LIN {X 30.043,Y -44.102,Z -90.850,A -90.000,B 90.000,C 0.000} C_DIS
LIN {X 31.596,Y -44.132,Z -91.106,A -90.000,B 90.000,C 0.000} C_DIS
LIN {X 31.805,Y -44.138,Z -91.148,A -90.000,B 90.000,C 0.000} C_DIS
LIN {X 31.963,Y -44.144,Z -91.180,A -90.000,B 90.000,C 0.000} C_DIS
LIN {X 32.126,Y -44.146,Z -91.221,A -90.000,B 90.000,C 0.000} C_DIS
LIN {X 33.590,Y -44.179,Z -91.628,A -90.000,B 90.000,C 0.000} C_DIS
LIN {X 33.752,Y -44.184,Z -91.677,A -90.000,B 90.000,C 0.000} C_DIS
LIN {X 33.947,Y -44.192,Z -91.742,A -90.000,B 90.000,C 0.000} C_DIS
LIN {X 34.606,Y -44.214,Z -91.970,A -90.000,B 90.000,C 0.000} C_DIS
LIN {X 35.661,Y -44.230,Z -92.339,A -90.000,B 90.000,C 0.000} C_DIS
LIN {X 35.939,Y -44.232,Z -92.438,A -90.000,B 90.000,C 0.000} C_DIS
LIN {X 36.161,Y -44.234,Z -92.528,A -90.000,B 90.000,C 0.000} C_DIS
LIN {X 36.724,Y -44.246,Z -92.772,A -90.000,B 90.000,C 0.000} C_DIS
LIN {X 36.900,Y -44.250,Z -92.851,A -90.000,B 90.000,C 0.000} C_DIS
LIN {X 37.063,Y -44.253,Z -92.930,A -90.000,B 90.000,C 0.000} C_DIS
LIN {X 37.996,Y -44.267,Z -93.435,A -90.000,B 90.000,C 0.000} C_DIS
LIN {X 38.705,Y -44.281,Z -93.837,A -90.000,B 90.000,C 0.000} C_DIS
LIN {X 39.137,Y -44.293,Z -94.082,A -90.000,B 90.000,C 0.000} C_DIS
LIN {X 39.281,Y -44.294,Z -94.165,A -90.000,B 90.000,C 0.000} C_DIS
LIN {X 39.455,Y -44.293,Z -94.272,A -90.000,B 90.000,C 0.000} C_DIS
LIN {X 40.133,Y -44.291,Z -94.711,A -90.000,B 90.000,C 0.000} C_DIS
LIN {X 40.366,Y -44.293,Z -94.872,A -90.000,B 90.000,C 0.000} C_DIS
LIN {X 40.619,Y -44.297,Z -95.057,A -90.000,B 90.000,C 0.000} C_DIS
LIN {X 40.830,Y -44.305,Z -95.230,A -90.000,B 90.000,C 0.000} C_DIS
LIN {X 41.144,Y -44.315,Z -95.490,A -90.000,B 90.000,C 0.000} C_DIS
LIN {X 41.855,Y -44.317,Z -96.085,A -90.000,B 90.000,C 0.000} C_DIS
LIN {X 42.021,Y -44.319,Z -96.232,A -90.000,B 90.000,C 0.000} C_DIS
LIN {X 42.450,Y -44.332,Z -96.645,A -90.000,B 90.000,C 0.000} C_DIS
LIN {X 42.787,Y -44.333,Z -96.974,A -90.000,B 90.000,C 0.000} C_DIS
LIN {X 42.967,Y -44.330,Z -97.150,A -90.000,B 90.000,C 0.000} C_DIS
LIN {X 43.705,Y -44.300,Z -97.883,A -90.000,B 90.000,C 0.000} C_DIS
LIN {X 43.789,Y -44.297,Z -97.971,A -90.000,B 90.000,C 0.000} C_DIS
LIN {X 44.031,Y -44.292,Z -98.239,A -90.000,B 90.000,C 0.000} C_DIS
LIN {X 44.098,Y -44.291,Z -98.318,A -90.000,B 90.000,C 0.000} C_DIS
LIN {X 44.222,Y -44.291,Z -98.469,A -90.000,B 90.000,C 0.000} C_DIS
LIN {X 44.387,Y -44.294,Z -98.687,A -90.000,B 90.000,C 0.000} C_DIS
LIN {X 44.481,Y -44.298,Z -98.827,A -90.000,B 90.000,C 0.000} C_DIS
LIN {X 44.610,Y -44.300,Z -99.041,A -90.000,B 90.000,C 0.000} C_DIS
LIN {X 44.729,Y -44.303,Z -99.246,A -90.000,B 90.000,C 0.000} C_DIS
LIN {X 45.134,Y -44.318,Z -99.976,A -90.000,B 90.000,C 0.000} C_DIS
LIN {X 45.262,Y -44.320,Z -100.209,A -90.000,B 90.000,C 0.000} C_DIS
LIN {X 45.761,Y -44.295,Z -101.133,A -90.000,B 90.000,C 0.000} C_DIS
LIN {X 45.808,Y -44.294,Z -101.226,A -90.000,B 90.000,C 0.000} C_DIS
LIN {X 46.111,Y -44.285,Z -101.863,A -90.000,B 90.000,C 0.000} C_DIS
LIN {X 46.252,Y -44.275,Z -102.164,A -90.000,B 90.000,C 0.000} C_DIS
LIN {X 46.732,Y -44.221,Z -103.202,A -90.000,B 90.000,C 0.000} C_DIS
LIN {X 46.781,Y -44.216,Z -103.318,A -90.000,B 90.000,C 0.000} C_DIS
LIN {X 46.871,Y -44.208,Z -103.549,A -90.000,B 90.000,C 0.000} C_DIS
LIN {X 46.913,Y -44.205,Z -103.666,A -90.000,B 90.000,C 0.000} C_DIS
LIN {X 46.986,Y -44.201,Z -103.892,A -90.000,B 90.000,C 0.000} C_DIS
LIN {X 47.046,Y -44.199,Z -104.098,A -90.000,B 90.000,C 0.000} C_DIS
LIN {X 47.095,Y -44.201,Z -104.309,A -90.000,B 90.000,C 0.000} C_DIS
LIN {X 47.115,Y -44.202,Z -104.397,A -90.000,B 90.000,C 0.000} C_DIS
LIN {X 47.180,Y -44.202,Z -104.648,A -90.000,B 90.000,C 0.000} C_DIS
LIN {X 47.223,Y -44.202,Z -104.839,A -90.000,B 90.000,C 0.000} C_DIS
LIN {X 47.252,Y -44.203,Z -104.996,A -90.000,B 90.000,C 0.000} C_DIS
LIN {X 47.278,Y -44.207,Z -105.181,A -90.000,B 90.000,C 0.000} C_DIS
LIN {X 47.321,Y -44.218,Z -105.570,A -90.000,B 90.000,C 0.000} C_DIS
LIN {X 47.363,Y -44.223,Z -106.056,A -90.000,B 90.000,C 0.000} C_DIS
LIN {X 47.384,Y -44.224,Z -106.317,A -90.000,B 90.000,C 0.000} C_DIS
LIN {X 47.440,Y -44.195,Z -107.093,A -90.000,B 90.000,C 0.000} C_DIS
LIN {X 47.552,Y -44.143,Z -108.663,A -90.000,B 90.000,C 0.000} C_DIS
LIN {X 47.559,Y -44.140,Z -108.785,A -90.000,B 90.000,C 0.000} C_DIS
LIN {X 47.562,Y -44.138,Z -108.944,A -90.000,B 90.000,C 0.000} C_DIS
LIN {X 47.556,Y -44.137,Z -109.182,A -90.000,B 90.000,C 0.000} C_DIS
LIN {X 47.550,Y -44.139,Z -109.300,A -90.000,B 90.000,C 0.000} C_DIS
LIN {X 47.472,Y -44.157,Z -110.305,A -90.000,B 90.000,C 0.000} C_DIS
LIN {X 47.309,Y -44.112,Z -112.094,A -90.000,B 90.000,C 0.000} C_DIS
LIN {X 47.205,Y -44.092,Z -113.075,A -90.000,B 90.000,C 0.000} C_DIS
LIN {X 47.187,Y -44.091,Z -113.203,A -90.000,B 90.000,C 0.000} C_DIS
LIN {X 47.137,Y -44.091,Z -113.498,A -90.000,B 90.000,C 0.000} C_DIS
LIN {X 47.119,Y -44.093,Z -113.585,A -90.000,B 90.000,C 0.000} C_DIS
LIN {X 47.045,Y -44.099,Z -113.899,A -90.000,B 90.000,C 0.000} C_DIS
LIN {X 46.943,Y -44.102,Z -114.328,A -90.000,B 90.000,C 0.000} C_DIS
LIN {X 46.601,Y -44.049,Z -115.684,A -90.000,B 90.000,C 0.000} C_DIS
LIN {X 46.560,Y -44.044,Z -115.831,A -90.000,B 90.000,C 0.000} C_DIS
LIN {X 46.147,Y -44.010,Z -117.234,A -90.000,B 90.000,C 0.000} C_DIS
LIN {X 46.088,Y -44.008,Z -117.419,A -90.000,B 90.000,C 0.000} C_DIS
LIN {X 45.995,Y -44.008,Z -117.676,A -90.000,B 90.000,C 0.000} C_DIS
LIN {X 45.962,Y -44.009,Z -117.763,A -90.000,B 90.000,C 0.000} C_DIS
LIN {X 45.889,Y -44.013,Z -117.937,A -90.000,B 90.000,C 0.000} C_DIS
LIN {X 45.762,Y -44.020,Z -118.219,A -90.000,B 90.000,C 0.000} C_DIS
LIN {X 45.357,Y -43.999,Z -119.084,A -90.000,B 90.000,C 0.000} C_DIS
LIN {X 45.158,Y -43.991,Z -119.498,A -90.000,B 90.000,C 0.000} C_DIS
LIN {X 44.451,Y -43.966,Z -120.974,A -90.000,B 90.000,C 0.000} C_DIS
LIN {X 44.317,Y -43.963,Z -121.251,A -90.000,B 90.000,C 0.000} C_DIS
LIN {X 44.210,Y -43.963,Z -121.454,A -90.000,B 90.000,C 0.000} C_DIS
LIN {X 44.078,Y -43.968,Z -121.683,A -90.000,B 90.000,C 0.000} C_DIS
LIN {X 43.957,Y -43.966,Z -121.881,A -90.000,B 90.000,C 0.000} C_DIS
LIN {X 43.022,Y -43.933,Z -123.308,A -90.000,B 90.000,C 0.000} C_DIS
LIN {X 42.446,Y -43.896,Z -124.174,A -90.000,B 90.000,C 0.000} C_DIS
LIN {X 42.367,Y -43.892,Z -124.288,A -90.000,B 90.000,C 0.000} C_DIS
LIN {X 41.848,Y -43.874,Z -125.016,A -90.000,B 90.000,C 0.000} C_DIS
LIN {X 41.755,Y -43.871,Z -125.141,A -90.000,B 90.000,C 0.000} C_DIS
LIN {X 40.950,Y -43.838,Z -126.136,A -90.000,B 90.000,C 0.000} C_DIS
LIN {X 40.132,Y -43.777,Z -127.128,A -90.000,B 90.000,C 0.000} C_DIS
LIN {X 39.865,Y -43.763,Z -127.435,A -90.000,B 90.000,C 0.000} C_DIS
LIN {X 39.099,Y -43.739,Z -128.268,A -90.000,B 90.000,C 0.000} C_DIS
LIN {X 38.728,Y -43.722,Z -128.669,A -90.000,B 90.000,C 0.000} C_DIS
LIN {X 38.085,Y -43.674,Z -129.350,A -90.000,B 90.000,C 0.000} C_DIS
LIN {X 37.439,Y -43.621,Z -130.031,A -90.000,B 90.000,C 0.000} C_DIS
LIN {X 37.295,Y -43.613,Z -130.175,A -90.000,B 90.000,C 0.000} C_DIS
LIN {X 36.203,Y -43.578,Z -131.197,A -90.000,B 90.000,C 0.000} C_DIS
LIN {X 35.591,Y -43.550,Z -131.813,A -90.000,B 90.000,C 0.000} C_DIS
LIN {X 34.765,Y -43.481,Z -132.619,A -90.000,B 90.000,C 0.000} C_DIS
LIN {X 34.182,Y -43.434,Z -133.184,A -90.000,B 90.000,C 0.000} C_DIS
LIN {X 34.040,Y -43.425,Z -133.315,A -90.000,B 90.000,C 0.000} C_DIS
LIN {X 32.759,Y -43.384,Z -134.425,A -90.000,B 90.000,C 0.000} C_DIS
LIN {X 31.780,Y -43.308,Z -135.363,A -90.000,B 90.000,C 0.000} C_DIS
LIN {X 31.780,Y -60.000,Z -135.363,A -90.000,B 90.000,C 0.000} C_DIS
LIN {X 27.880,Y -60.000,Z -88.546,A -90.000,B 90.000,C 0.000} C_DIS
LIN {X 27.880,Y -43.308,Z -88.546,A -90.000,B 90.000,C 0.000} C_DIS
LIN {X 28.059,Y -43.318,Z -88.565,A -90.000,B 90.000,C 0.000} C_DIS
LIN {X 28.163,Y -43.325,Z -88.579,A -90.000,B 90.000,C 0.000} C_DIS
LIN {X 28.312,Y -43.338,Z -88.598,A -90.000,B 90.000,C 0.000} C_DIS
LIN {X 28.537,Y -43.361,Z -88.634,A -90.000,B 90.000,C 0.000} C_DIS
LIN {X 29.638,Y -43.432,Z -88.839,A -90.000,B 90.000,C 0.000} C_DIS
LIN {X 30.344,Y -43.470,Z -88.974,A -90.000,B 90.000,C 0.000} C_DIS
LIN {X 30.370,Y -43.472,Z -88.979,A -90.000,B 90.000,C 0.000} C_DIS
LIN {X 31.919,Y -43.541,Z -89.223,A -90.000,B 90.000,C 0.000} C_DIS
LIN {X 32.192,Y -43.555,Z -89.274,A -90.000,B 90.000,C 0.000} C_DIS
LIN {X 32.370,Y -43.563,Z -89.310,A -90.000,B 90.000,C 0.000} C_DIS
LIN {X 32.600,Y -43.574,Z -89.365,A -90.000,B 90.000,C 0.000} C_DIS
LIN {X 34.122,Y -43.639,Z -89.777,A -90.000,B 90.000,C 0.000} C_DIS
LIN {X 34.326,Y -43.649,Z -89.837,A -90.000,B 90.000,C 0.000} C_DIS
LIN {X 34.574,Y -43.663,Z -89.918,A -90.000,B 90.000,C 0.000} C_DIS
LIN {X 34.743,Y -43.669,Z -89.976,A -90.000,B 90.000,C 0.000} C_DIS
LIN {X 36.312,Y -43.705,Z -90.522,A -90.000,B 90.000,C 0.000} C_DIS
LIN {X 36.590,Y -43.708,Z -90.621,A -90.000,B 90.000,C 0.000} C_DIS
LIN {X 36.883,Y -43.714,Z -90.736,A -90.000,B 90.000,C 0.000} C_DIS
LIN {X 37.249,Y -43.714,Z -90.897,A -90.000,B 90.000,C 0.000} C_DIS
LIN {X 37.752,Y -43.711,Z -91.123,A -90.000,B 90.000,C 0.000} C_DIS
LIN {X 37.986,Y -43.719,Z -91.238,A -90.000,B 90.000,C 0.000} C_DIS
LIN {X 38.913,Y -43.761,Z -91.731,A -90.000,B 90.000,C 0.000} C_DIS
LIN {X 38.987,Y -43.763,Z -91.772,A -90.000,B 90.000,C 0.000} C_DIS
LIN {X 39.920,Y -43.783,Z -92.302,A -90.000,B 90.000,C 0.000} C_DIS
LIN {X 40.246,Y -43.784,Z -92.489,A -90.000,B 90.000,C 0.000} C_DIS
LIN {X 40.465,Y -43.786,Z -92.621,A -90.000,B 90.000,C 0.000} C_DIS
LIN {X 40.951,Y -43.795,Z -92.932,A -90.000,B 90.000,C 0.000} C_DIS
LIN {X 41.185,Y -43.792,Z -93.085,A -90.000,B 90.000,C 0.000} C_DIS
LIN {X 41.470,Y -43.790,Z -93.283,A -90.000,B 90.000,C 0.000} C_DIS
LIN {X 41.766,Y -43.790,Z -93.499,A -90.000,B 90.000,C 0.000} C_DIS
LIN {X 41.857,Y -43.790,Z -93.570,A -90.000,B 90.000,C 0.000} C_DIS
LIN {X 42.397,Y -43.801,Z -94.019,A -90.000,B 90.000,C 0.000} C_DIS
LIN {X 42.561,Y -43.807,Z -94.153,A -90.000,B 90.000,C 0.000} C_DIS
LIN {X 42.874,Y -43.816,Z -94.412,A -90.000,B 90.000,C 0.000} C_DIS
LIN {X 43.145,Y -43.817,Z -94.640,A -90.000,B 90.000,C 0.000} C_DIS
LIN {X 43.339,Y -43.815,Z -94.815,A -90.000,B 90.000,C 0.000} C_DIS
LIN {X 44.418,Y -43.818,Z -95.866,A -90.000,B 90.000,C 0.000} C_DIS
LIN {X 44.651,Y -43.815,Z -96.094,A -90.000,B 90.000,C 0.000} C_DIS
LIN {X 45.058,Y -43.797,Z -96.498,A -90.000,B 90.000,C 0.000} C_DIS
LIN {X 45.182,Y -43.793,Z -96.627,A -90.000,B 90.000,C 0.000} C_DIS
LIN {X 45.463,Y -43.786,Z -96.938,A -90.000,B 90.000,C 0.000} C_DIS
LIN {X 45.596,Y -43.784,Z -97.094,A -90.000,B 90.000,C 0.000} C_DIS
LIN {X 45.754,Y -43.783,Z -97.288,A -90.000,B 90.000,C 0.000} C_DIS
LIN {X 45.968,Y -43.786,Z -97.573,A -90.000,B 90.000,C 0.000} C_DIS
LIN {X 46.087,Y -43.783,Z -97.752,A -90.000,B 90.000,C 0.000} C_DIS
LIN {X 46.267,Y -43.781,Z -98.049,A -90.000,B 90.000,C 0.000} C_DIS
LIN {X 46.405,Y -43.780,Z -98.288,A -90.000,B 90.000,C 0.000} C_DIS
LIN {X 47.442,Y -43.730,Z -100.210,A -90.000,B 90.000,C 0.000} C_DIS
LIN {X 47.514,Y -43.727,Z -100.349,A -90.000,B 90.000,C 0.000} C_DIS
LIN {X 48.139,Y -43.712,Z -101.661,A -90.000,B 90.000,C 0.000} C_DIS
LIN {X 48.380,Y -43.693,Z -102.177,A -90.000,B 90.000,C 0.000} C_DIS
LIN {X 48.470,Y -43.682,Z -102.371,A -90.000,B 90.000,C 0.000} C_DIS
LIN {X 48.568,Y -43.669,Z -102.606,A -90.000,B 90.000,C 0.000} C_DIS
LIN {X 48.643,Y -43.653,Z -102.804,A -90.000,B 90.000,C 0.000} C_DIS
LIN {X 48.715,Y -43.636,Z -103.011,A -90.000,B 90.000,C 0.000} C_DIS
LIN {X 48.803,Y -43.616,Z -103.296,A -90.000,B 90.000,C 0.000} C_DIS
LIN {X 48.876,Y -43.601,Z -103.555,A -90.000,B 90.000,C 0.000} C_DIS
LIN {X 48.905,Y -43.595,Z -103.673,A -90.000,B 90.000,C 0.000} C_DIS
LIN {X 48.958,Y -43.586,Z -103.919,A -90.000,B 90.000,C 0.000} C_DIS
LIN {X 49.017,Y -43.574,Z -104.168,A -90.000,B 90.000,C 0.000} C_DIS
LIN {X 49.083,Y -43.562,Z -104.475,A -90.000,B 90.000,C 0.000} C_DIS
LIN {X 49.116,Y -43.558,Z -104.663,A -90.000,B 90.000,C 0.000} C_DIS
LIN {X 49.152,Y -43.556,Z -104.928,A -90.000,B 90.000,C 0.000} C_DIS
LIN {X 49.200,Y -43.558,Z -105.382,A -90.000,B 90.000,C 0.000} C_DIS
LIN {X 49.314,Y -43.572,Z -106.702,A -90.000,B 90.000,C 0.000} C_DIS
LIN {X 49.338,Y -43.572,Z -106.983,A -90.000,B 90.000,C 0.000} C_DIS
LIN {X 49.445,Y -43.516,Z -108.506,A -90.000,B 90.000,C 0.000} C_DIS
LIN {X 49.454,Y -43.501,Z -108.743,A -90.000,B 90.000,C 0.000} C_DIS
LIN {X 49.455,Y -43.493,Z -108.912,A -90.000,B 90.000,C 0.000} C_DIS
LIN {X 49.446,Y -43.483,Z -109.215,A -90.000,B 90.000,C 0.000} C_DIS
LIN {X 49.435,Y -43.479,Z -109.402,A -90.000,B 90.000,C 0.000} C_DIS
LIN {X 49.294,Y -43.461,Z -111.026,A -90.000,B 90.000,C 0.000} C_DIS
LIN {X 49.267,Y -43.452,Z -111.313,A -90.000,B 90.000,C 0.000} C_DIS
LIN {X 49.173,Y -43.402,Z -112.245,A -90.000,B 90.000,C 0.000} C_DIS
LIN {X 49.055,Y -43.354,Z -113.257,A -90.000,B 90.000,C 0.000} C_DIS
LIN {X 49.016,Y -43.344,Z -113.516,A -90.000,B 90.000,C 0.000} C_DIS
LIN {X 48.949,Y -43.336,Z -113.881,A -90.000,B 90.000,C 0.000} C_DIS
LIN {X 48.918,Y -43.336,Z -114.020,A -90.000,B 90.000,C 0.000} C_DIS
LIN {X 48.648,Y -43.340,Z -115.154,A -90.000,B 90.000,C 0.000} C_DIS
LIN {X 48.456,Y -43.308,Z -115.911,A -90.000,B 90.000,C 0.000} C_DIS
LIN {X 48.456,Y -60.000,Z -115.911,A -90.000,B 90.000,C 0.000} C_DIS
LIN {X 43.124,Y -60.000,Z -92.100,A -90.000,B 90.000,C 0.000} C_DIS
LIN {X 43.124,Y -43.308,Z -92.100,A -90.000,B 90.000,C 0.000} C_DIS
LIN {X 43.760,Y -43.320,Z -92.627,A -90.000,B 90.000,C 0.000} C_DIS
LIN {X 44.439,Y -43.322,Z -93.197,A -90.000,B 90.000,C 0.000} C_DIS
LIN {X 44.570,Y -43.324,Z -93.315,A -90.000,B 90.000,C 0.000} C_DIS
LIN {X 44.698,Y -43.320,Z -93.434,A -90.000,B 90.000,C 0.000} C_DIS
LIN {X 45.276,Y -43.308,Z -94.001,A -90.000,B 90.000,C 0.000} C_DIS
LIN {X 45.276,Y -60.000,Z -94.001,A -90.000,B 90.000,C 0.000} C_DIS
LIN {X -15.244,Y -60.000,Z -137.680,A -90.000,B 90.000,C 0.000} C_DIS
LIN {X -15.244,Y -43.308,Z -137.680,A -90.000,B 90.000,C 0.000} C_DIS
LIN {X -15.380,Y -43.347,Z -137.361,A -90.000,B 90.000,C 0.000} C_DIS
LIN {X -15.513,Y -43.390,Z -137.028,A -90.000,B 90.000,C 0.000} C_DIS
LIN {X -15.611,Y -43.411,Z -136.767,A -90.000,B 90.000,C 0.000} C_DIS
LIN {X -15.839,Y -43.449,Z -136.149,A -90.000,B 90.000,C 0.000} C_DIS
LIN {X -15.880,Y -43.453,Z -136.030,A -90.000,B 90.000,C 0.000} C_DIS
LIN {X -16.000,Y -43.464,Z -135.661,A -90.000,B 90.000,C 0.000} C_DIS
LIN {X -16.068,Y -43.474,Z -135.427,A -90.000,B 90.000,C 0.000} C_DIS
LIN {X -16.120,Y -43.485,Z -135.220,A -90.000,B 90.000,C 0.000} C_DIS
LIN {X -16.156,Y -43.495,Z -135.060,A -90.000,B 90.000,C 0.000} C_DIS
LIN {X -16.243,Y -43.528,Z -134.606,A -90.000,B 90.000,C 0.000} C_DIS
LIN {X -16.291,Y -43.540,Z -134.342,A -90.000,B 90.000,C 0.000} C_DIS
LIN {X -16.453,Y -43.560,Z -133.399,A -90.000,B 90.000,C 0.000} C_DIS
LIN {X -16.487,Y -43.566,Z -133.170,A -90.000,B 90.000,C 0.000} C_DIS
LIN {X -16.536,Y -43.579,Z -132.789,A -90.000,B 90.000,C 0.000} C_DIS
LIN {X -16.555,Y -43.590,Z -132.587,A -90.000,B 90.000,C 0.000} C_DIS
LIN {X -16.567,Y -43.598,Z -132.329,A -90.000,B 90.000,C 0.000} C_DIS
LIN {X -16.575,Y -43.608,Z -132.021,A -90.000,B 90.000,C 0.000} C_DIS
LIN {X -16.575,Y -43.613,Z -131.842,A -90.000,B 90.000,C 0.000} C_DIS
LIN {X -16.565,Y -43.622,Z -131.524,A -90.000,B 90.000,C 0.000} C_DIS
LIN {X -16.533,Y -43.637,Z -131.071,A -90.000,B 90.000,C 0.000} C_DIS
LIN {X -16.510,Y -43.647,Z -130.766,A -90.000,B 90.000,C 0.000} C_DIS
LIN {X -16.464,Y -43.666,Z -130.269,A -90.000,B 90.000,C 0.000} C_DIS
LIN {X -16.339,Y -43.680,Z -129.038,A -90.000,B 90.000,C 0.000} C_DIS
LIN {X -16.304,Y -43.685,Z -128.769,A -90.000,B 90.000,C 0.000} C_DIS
LIN {X -16.269,Y -43.692,Z -128.557,A -90.000,B 90.000,C 0.000} C_DIS
LIN {X -16.232,Y -43.701,Z -128.334,A -90.000,B 90.000,C 0.000} C_DIS
LIN {X -16.080,Y -43.723,Z -127.467,A -90.000,B 90.000,C 0.000} C_DIS
LIN {X -16.014,Y -43.733,Z -127.175,A -90.000,B 90.000,C 0.000} C_DIS
LIN {X -15.964,Y -43.742,Z -126.978,A -90.000,B 90.000,C 0.000} C_DIS
LIN {X -15.876,Y -43.758,Z -126.673,A -90.000,B 90.000,C 0.000} C_DIS
LIN {X -15.607,Y -43.810,Z -125.802,A -90.000,B 90.000,C 0.000} C_DIS
LIN {X -15.423,Y -43.845,Z -125.098,A -90.000,B 90.000,C 0.000} C_DIS
LIN {X -15.140,Y -43.879,Z -124.031,A -90.000,B 90.000,C 0.000} C_DIS
LIN {X -15.107,Y -43.886,Z -123.903,A -90.000,B 90.000,C 0.000} C_DIS
LIN {X -15.003,Y -43.907,Z -123.535,A -90.000,B 90.000,C 0.000} C_DIS
LIN {X -14.926,Y -43.923,Z -123.288,A -90.000,B 90.000,C 0.000} C_DIS
LIN {X -14.894,Y -43.930,Z -123.197,A -90.000,B 90.000,C 0.000} C_DIS
LIN {X -14.591,Y -43.993,Z -122.282,A -90.000,B 90.000,C 0.000} C_DIS
LIN {X -14.514,Y -44.006,Z -122.051,A -90.000,B 90.000,C 0.000} C_DIS
LIN {X -14.440,Y -44.014,Z -121.831,A -90.000,B 90.000,C 0.000} C_DIS
LIN {X -14.308,Y -44.042,Z -121.432,A -90.000,B 90.000,C 0.000} C_DIS
LIN {X -14.269,Y -44.055,Z -121.204,A -90.000,B 90.000,C 0.000} C_DIS
LIN {X -14.224,Y -44.068,Z -120.986,A -90.000,B 90.000,C 0.000} C_DIS
LIN {X -14.177,Y -44.081,Z -120.781,A -90.000,B 90.000,C 0.000} C_DIS
LIN {X -14.137,Y -44.092,Z -120.621,A -90.000,B 90.000,C 0.000} C_DIS
LIN {X -14.049,Y -44.115,Z -120.313,A -90.000,B 90.000,C 0.000} C_DIS
LIN {X -14.009,Y -44.125,Z -120.190,A -90.000,B 90.000,C 0.000} C_DIS
LIN {X -13.914,Y -44.149,Z -119.908,A -90.000,B 90.000,C 0.000} C_DIS
LIN {X -13.658,Y -44.210,Z -119.226,A -90.000,B 90.000,C 0.000} C_DIS
LIN {X -13.526,Y -44.246,Z -118.874,A -90.000,B 90.000,C 0.000} C_DIS
LIN {X -13.483,Y -44.265,Z -118.568,A -90.000,B 90.000,C 0.000} C_DIS
LIN {X -13.412,Y -44.290,Z -118.074,A -90.000,B 90.000,C 0.000} C_DIS
LIN {X -13.383,Y -44.299,Z -117.901,A -90.000,B 90.000,C 0.000} C_DIS
LIN {X -13.308,Y -44.320,Z -117.527,A -90.000,B 90.000,C 0.000} C_DIS
LIN {X -13.271,Y -44.330,Z -117.366,A -90.000,B 90.000,C 0.000} C_DIS
LIN {X -13.199,Y -44.348,Z -117.097,A -90.000,B 90.000,C 0.000} C_DIS
LIN {X -13.117,Y -44.368,Z -116.835,A -90.000,B 90.000,C 0.000} C_DIS
LIN {X -13.068,Y -44.391,Z -116.236,A -90.000,B 90.000,C 0.000} C_DIS
LIN {X -13.054,Y -44.401,Z -116.062,A -90.000,B 90.000,C 0.000} C_DIS
LIN {X -13.025,Y -44.417,Z -115.794,A -90.000,B 90.000,C 0.000} C_DIS
LIN {X -13.027,Y -44.433,Z -115.413,A -90.000,B 90.000,C 0.000} C_DIS
LIN {X -13.025,Y -44.437,Z -115.311,A -90.000,B 90.000,C 0.000} C_DIS
LIN {X -12.980,Y -44.485,Z -114.346,A -90.000,B 90.000,C 0.000} C_DIS
LIN {X -12.971,Y -44.492,Z -114.160,A -90.000,B 90.000,C 0.000} C_DIS
LIN {X -13.096,Y -44.488,Z -113.713,A -90.000,B 90.000,C 0.000} C_DIS
LIN {X -13.142,Y -44.487,Z -113.531,A -90.000,B 90.000,C 0.000} C_DIS
LIN {X -13.209,Y -44.487,Z -113.225,A -90.000,B 90.000,C 0.000} C_DIS
LIN {X -13.247,Y -44.487,Z -113.025,A -90.000,B 90.000,C 0.000} C_DIS
LIN {X -13.270,Y -44.489,Z -112.861,A -90.000,B 90.000,C 0.000} C_DIS
LIN {X -13.279,Y -44.488,Z -112.843,A -90.000,B 90.000,C 0.000} C_DIS
LIN {X -13.339,Y -44.484,Z -112.702,A -90.000,B 90.000,C 0.000} C_DIS
LIN {X -13.422,Y -44.479,Z -112.491,A -90.000,B 90.000,C 0.000} C_DIS
LIN {X -13.524,Y -44.481,Z -112.210,A -90.000,B 90.000,C 0.000} C_DIS
LIN {X -13.626,Y -44.484,Z -111.893,A -90.000,B 90.000,C 0.000} C_DIS
LIN {X -13.795,Y -44.487,Z -111.327,A -90.000,B 90.000,C 0.000} C_DIS
LIN {X -13.914,Y -44.481,Z -111.079,A -90.000,B 90.000,C 0.000} C_DIS
LIN {X -13.999,Y -44.477,Z -110.897,A -90.000,B 90.000,C 0.000} C_DIS
LIN {X -14.056,Y -44.475,Z -110.766,A -90.000,B 90.000,C 0.000} C_DIS
LIN {X -14.266,Y -44.470,Z -110.237,A -90.000,B 90.000,C 0.000} C_DIS
LIN {X -14.549,Y -44.474,Z -109.519,A -90.000,B 90.000,C 0.000} C_DIS
LIN {X -14.678,Y -44.470,Z -109.274,A -90.000,B 90.000,C 0.000} C_DIS
LIN {X -15.006,Y -44.456,Z -108.656,A -90.000,B 90.000,C 0.000} C_DIS
LIN {X -15.402,Y -44.440,Z -107.909,A -90.000,B 90.000,C 0.000} C_DIS
LIN {X -15.440,Y -44.439,Z -107.833,A -90.000,B 90.000,C 0.000} C_DIS
LIN {X -15.512,Y -44.438,Z -107.685,A -90.000,B 90.000,C 0.000} C_DIS
LIN {X -15.616,Y -44.438,Z -107.452,A -90.000,B 90.000,C 0.000} C_DIS
LIN {X -15.691,Y -44.438,Z -107.273,A -90.000,B 90.000,C 0.000} C_DIS
LIN {X -15.833,Y -44.441,Z -106.901,A -90.000,B 90.000,C 0.000} C_DIS
LIN {X -15.976,Y -44.446,Z -106.496,A -90.000,B 90.000,C 0.000} C_DIS
LIN {X -16.349,Y -44.442,Z -105.430,A -90.000,B 90.000,C 0.000} C_DIS
LIN {X -16.573,Y -44.435,Z -104.785,A -90.000,B 90.000,C 0.000} C_DIS
LIN {X -16.645,Y -44.433,Z -104.573,A -90.000,B 90.000,C 0.000} C_DIS
LIN {X -16.697,Y -44.432,Z -104.408,A -90.000,B 90.000,C 0.000} C_DIS
LIN {X -16.897,Y -44.431,Z -103.683,A -90.000,B 90.000,C 0.000} C_DIS
LIN {X -17.066,Y -44.429,Z -103.059,A -90.000,B 90.000,C 0.000} C_DIS
LIN {X -17.108,Y -44.429,Z -102.880,A -90.000,B 90.000,C 0.000} C_DIS
LIN {X -17.163,Y -44.431,Z -102.601,A -90.000,B 90.000,C 0.000} C_DIS
LIN {X -17.192,Y -44.433,Z -102.425,A -90.000,B 90.000,C 0.000} C_DIS
LIN {X -17.220,Y -44.438,Z -102.198,A -90.000,B 90.000,C 0.000} C_DIS
LIN {X -17.301,Y -44.444,Z -101.509,A -90.000,B 90.000,C 0.000} C_DIS
LIN {X -17.425,Y -44.437,Z -100.434,A -90.000,B 90.000,C 0.000} C_DIS
LIN {X -17.473,Y -44.433,Z -100.202,A -90.000,B 90.000,C 0.000} C_DIS
LIN {X -17.537,Y -44.428,Z -99.815,A -90.000,B 90.000,C 0.000} C_DIS
LIN {X -17.564,Y -44.426,Z -99.576,A -90.000,B 90.000,C 0.000} C_DIS
LIN {X -17.584,Y -44.423,Z -99.289,A -90.000,B 90.000,C 0.000} C_DIS
LIN {X -17.590,Y -44.420,Z -99.195,A -90.000,B 90.000,C 0.000} C_DIS
LIN {X -17.595,Y -44.411,Z -98.998,A -90.000,B 90.000,C 0.000} C_DIS
LIN {X -17.593,Y -44.396,Z -98.704,A -90.000,B 90.000,C 0.000} C_DIS
LIN {X -17.587,Y -44.391,Z -98.555,A -90.000,B 90.000,C 0.000} C_DIS
LIN {X -17.565,Y -44.382,Z -98.281,A -90.000,B 90.000,C 0.000} C_DIS
LIN {X -17.556,Y -44.380,Z -98.195,A -90.000,B 90.000,C 0.000} C_DIS
LIN {X -17.489,Y -44.372,Z -97.744,A -90.000,B 90.000,C 0.000} C_DIS
LIN {X -17.457,Y -44.370,Z -97.581,A -90.000,B 90.000,C 0.000} C_DIS
LIN {X -17.379,Y -44.369,Z -97.241,A -90.000,B 90.000,C 0.000} C_DIS
LIN {X -17.346,Y -44.369,Z -97.114,A -90.000,B 90.000,C 0.000} C_DIS
LIN {X -17.205,Y -44.373,Z -96.624,A -90.000,B 90.000,C 0.000} C_DIS
LIN {X -17.153,Y -44.366,Z -96.453,A -90.000,B 90.000,C 0.000} C_DIS
LIN {X -16.994,Y -44.336,Z -95.932,A -90.000,B 90.000,C 0.000} C_DIS
LIN {X -16.781,Y -44.305,Z -95.224,A -90.000,B 90.000,C 0.000} C_DIS
LIN {X -16.677,Y -44.293,Z -94.911,A -90.000,B 90.000,C 0.000} C_DIS
LIN {X -16.494,Y -44.277,Z -94.416,A -90.000,B 90.000,C 0.000} C_DIS
LIN {X -16.461,Y -44.275,Z -94.332,A -90.000,B 90.000,C 0.000} C_DIS
LIN {X -16.368,Y -44.270,Z -94.113,A -90.000,B 90.000,C 0.000} C_DIS
LIN {X -16.272,Y -44.257,Z -93.910,A -90.000,B 90.000,C 0.000} C_DIS
LIN {X -16.201,Y -44.247,Z -93.776,A -90.000,B 90.000,C 0.000} C_DIS
LIN {X -16.083,Y -44.231,Z -93.560,A -90.000,B 90.000,C 0.000} C_DIS
LIN {X -15.965,Y -44.217,Z -93.360,A -90.000,B 90.000,C 0.000} C_DIS
LIN {X -15.901,Y -44.211,Z -93.261,A -90.000,B 90.000,C 0.000} C_DIS
LIN {X -15.689,Y -44.196,Z -92.938,A -90.000,B 90.000,C 0.000} C_DIS
LIN {X -15.529,Y -44.189,Z -92.725,A -90.000,B 90.000,C 0.000} C_DIS
LIN {X -15.350,Y -44.185,Z -92.508,A -90.000,B 90.000,C 0.000} C_DIS
LIN {X -14.962,Y -44.180,Z -92.068,A -90.000,B 90.000,C 0.000} C_DIS
LIN {X -14.790,Y -44.179,Z -91.883,A -90.000,B 90.000,C 0.000} C_DIS
LIN {X -14.638,Y -44.171,Z -91.724,A -90.000,B 90.000,C 0.000} C_DIS
LIN {X -13.817,Y -44.113,Z -90.872,A -90.000,B 90.000,C 0.000} C_DIS
LIN {X -13.699,Y -44.100,Z -90.729,A -90.000,B 90.000,C 0.000} C_DIS
LIN {X -13.563,Y -44.088,Z -90.577,A -90.000,B 90.000,C 0.000} C_DIS
LIN {X -13.373,Y -44.074,Z -90.379,A -90.000,B 90.000,C 0.000} C_DIS
LIN {X -13.214,Y -44.064,Z -90.221,A -90.000,B 90.000,C 0.000} C_DIS
LIN {X -12.987,Y -44.052,Z -90.010,A -90.000,B 90.000,C 0.000} C_DIS
LIN {X -12.902,Y -44.049,Z -89.936,A -90.000,B 90.000,C 0.000} C_DIS
LIN {X -12.746,Y -44.044,Z -89.808,A -90.000,B 90.000,C 0.000} C_DIS
LIN {X -12.680,Y -44.043,Z -89.758,A -90.000,B 90.000,C 0.000} C_DIS
LIN {X -12.573,Y -44.038,Z -89.677,A -90.000,B 90.000,C 0.000} C_DIS
LIN {X -12.331,Y -44.025,Z -89.510,A -90.000,B 90.000,C 0.000} C_DIS
LIN {X -12.210,Y -44.019,Z -89.432,A -90.000,B 90.000,C 0.000} C_DIS
LIN {X -11.699,Y -43.997,Z -89.125,A -90.000,B 90.000,C 0.000} C_DIS
LIN {X -11.423,Y -43.987,Z -88.973,A -90.000,B 90.000,C 0.000} C_DIS
LIN {X -10.162,Y -43.953,Z -88.327,A -90.000,B 90.000,C 0.000} C_DIS
LIN {X -9.975,Y -43.944,Z -88.233,A -90.000,B 90.000,C 0.000} C_DIS
LIN {X -9.414,Y -43.915,Z -87.946,A -90.000,B 90.000,C 0.000} C_DIS
LIN {X -9.268,Y -43.903,Z -87.872,A -90.000,B 90.000,C 0.000} C_DIS
LIN {X -8.463,Y -43.840,Z -87.465,A -90.000,B 90.000,C 0.000} C_DIS
LIN {X -8.390,Y -43.835,Z -87.430,A -90.000,B 90.000,C 0.000} C_DIS
LIN {X -8.075,Y -43.815,Z -87.289,A -90.000,B 90.000,C 0.000} C_DIS
LIN {X -7.871,Y -43.804,Z -87.205,A -90.000,B 90.000,C 0.000} C_DIS
LIN {X -7.688,Y -43.797,Z -87.138,A -90.000,B 90.000,C 0.000} C_DIS
LIN {X -7.471,Y -43.783,Z -87.064,A -90.000,B 90.000,C 0.000} C_DIS
LIN {X -7.307,Y -43.772,Z -87.009,A -90.000,B 90.000,C 0.000} C_DIS
LIN {X -7.194,Y -43.767,Z -86.977,A -90.000,B 90.000,C 0.000} C_DIS
LIN {X -6.071,Y -43.718,Z -86.685,A -90.000,B 90.000,C 0.000} C_DIS
LIN {X -5.656,Y -43.705,Z -86.591,A -90.000,B 90.000,C 0.000} C_DIS
LIN {X -5.225,Y -43.695,Z -86.507,A -90.000,B 90.000,C 0.000} C_DIS
LIN {X -4.857,Y -43.683,Z -86.438,A -90.000,B 90.000,C 0.000} C_DIS
LIN {X -4.394,Y -43.661,Z -86.353,A -90.000,B 90.000,C 0.000} C_DIS
LIN {X -4.258,Y -43.652,Z -86.329,A -90.000,B 90.000,C 0.000} C_DIS
LIN {X -3.948,Y -43.633,Z -86.277,A -90.000,B 90.000,C 0.000} C_DIS
LIN {X -2.427,Y -43.557,Z -86.072,A -90.000,B 90.000,C 0.000} C_DIS
LIN {X -2.075,Y -43.542,Z -86.037,A -90.000,B 90.000,C 0.000} C_DIS
LIN {X -0.953,Y -43.475,Z -85.939,A -90.000,B 90.000,C 0.000} C_DIS
LIN {X -0.675,Y -43.461,Z -85.922,A -90.000,B 90.000,C 0.000} C_DIS
LIN {X -0.002,Y -43.434,Z -85.905,A -90.000,B 90.000,C 0.000} C_DIS
LIN {X 0.610,Y -43.412,Z -85.888,A -90.000,B 90.000,C 0.000} C_DIS
LIN {X 0.846,Y -43.404,Z -85.884,A -90.000,B 90.000,C 0.000} C_DIS
LIN {X 1.330,Y -43.382,Z -85.881,A -90.000,B 90.000,C 0.000} C_DIS
LIN {X 1.593,Y -43.371,Z -85.884,A -90.000,B 90.000,C 0.000} C_DIS
LIN {X 1.841,Y -43.363,Z -85.894,A -90.000,B 90.000,C 0.000} C_DIS
LIN {X 2.166,Y -43.351,Z -85.909,A -90.000,B 90.000,C 0.000} C_DIS
LIN {X 3.538,Y -43.308,Z -86.008,A -90.000,B 90.000,C 0.000} C_DIS
LIN {X 3.538,Y -60.000,Z -86.008,A -90.000,B 90.000,C 0.000} C_DIS
LIN {X -17.683,Y -60.000,Z -125.925,A -90.000,B 90.000,C 0.000} C_DIS
LIN {X -17.683,Y -43.308,Z -125.925,A -90.000,B 90.000,C 0.000} C_DIS
LIN {X -17.472,Y -43.351,Z -125.245,A -90.000,B 90.000,C 0.000} C_DIS
LIN {X -17.378,Y -43.369,Z -124.883,A -90.000,B 90.000,C 0.000} C_DIS
LIN {X -17.247,Y -43.407,Z -124.368,A -90.000,B 90.000,C 0.000} C_DIS
LIN {X -17.092,Y -43.463,Z -123.754,A -90.000,B 90.000,C 0.000} C_DIS
LIN {X -16.979,Y -43.499,Z -123.316,A -90.000,B 90.000,C 0.000} C_DIS
LIN {X -16.893,Y -43.524,Z -123.003,A -90.000,B 90.000,C 0.000} C_DIS
LIN {X -16.794,Y -43.552,Z -122.679,A -90.000,B 90.000,C 0.000} C_DIS
LIN {X -16.446,Y -43.646,Z -121.620,A -90.000,B 90.000,C 0.000} C_DIS
LIN {X -16.222,Y -43.708,Z -120.935,A -90.000,B 90.000,C 0.000} C_DIS
LIN {X -16.208,Y -43.714,Z -120.851,A -90.000,B 90.000,C 0.000} C_DIS
LIN {X -16.151,Y -43.735,Z -120.568,A -90.000,B 90.000,C 0.000} C_DIS
LIN {X -16.108,Y -43.750,Z -120.375,A -90.000,B 90.000,C 0.000} C_DIS
LIN {X -16.050,Y -43.770,Z -120.137,A -90.000,B 90.000,C 0.000} C_DIS
LIN {X -15.985,Y -43.791,Z -119.899,A -90.000,B 90.000,C 0.000} C_DIS
LIN {X -15.915,Y -43.812,Z -119.662,A -90.000,B 90.000,C 0.000} C_DIS
LIN {X -15.780,Y -43.851,Z -119.252,A -90.000,B 90.000,C 0.000} C_DIS
LIN {X -15.446,Y -43.932,Z -118.360,A -90.000,B 90.000,C 0.000} C_DIS
LIN {X -15.390,Y -43.954,Z -117.965,A -90.000,B 90.000,C 0.000} C_DIS
LIN {X -15.351,Y -43.971,Z -117.699,A -90.000,B 90.000,C 0.000} C_DIS
LIN {X -15.327,Y -43.981,Z -117.557,A -90.000,B 90.000,C 0.000} C_DIS
LIN {X -15.254,Y -44.008,Z -117.180,A -90.000,B 90.000,C 0.000} C_DIS
LIN {X -15.195,Y -44.029,Z -116.911,A -90.000,B 90.000,C 0.000} C_DIS
LIN {X -15.105,Y -44.058,Z -116.565,A -90.000,B 90.000,C 0.000} C_DIS
LIN {X -15.067,Y -44.069,Z -116.438,A -90.000,B 90.000,C 0.000} C_DIS
LIN {X -15.023,Y -44.098,Z -115.889,A -90.000,B 90.000,C 0.000} C_DIS
LIN {X -15.001,Y -44.110,Z -115.677,A -90.000,B 90.000,C 0.000} C_DIS
LIN {X -15.002,Y -44.118,Z -115.441,A -90.000,B 90.000,C 0.000} C_DIS
LIN {X -14.999,Y -44.123,Z -115.255,A -90.000,B 90.000,C 0.000} C_DIS
LIN {X -14.959,Y -44.167,Z -114.380,A -90.000,B 90.000,C 0.000} C_DIS
LIN {X -14.991,Y -44.167,Z -114.267,A -90.000,B 90.000,C 0.000} C_DIS
LIN {X -15.056,Y -44.170,Z -114.018,A -90.000,B 90.000,C 0.000} C_DIS
LIN {X -15.139,Y -44.176,Z -113.647,A -90.000,B 90.000,C 0.000} C_DIS
LIN {X -15.186,Y -44.180,Z -113.407,A -90.000,B 90.000,C 0.000} C_DIS
LIN {X -15.260,Y -44.179,Z -113.221,A -90.000,B 90.000,C 0.000} C_DIS
LIN {X -15.383,Y -44.177,Z -112.881,A -90.000,B 90.000,C 0.000} C_DIS
LIN {X -15.500,Y -44.177,Z -112.522,A -90.000,B 90.000,C 0.000} C_DIS
LIN {X -15.643,Y -44.179,Z -112.044,A -90.000,B 90.000,C 0.000} C_DIS
LIN {X -15.788,Y -44.173,Z -111.739,A -90.000,B 90.000,C 0.000} C_DIS
LIN {X -15.892,Y -44.169,Z -111.497,A -90.000,B 90.000,C 0.000} C_DIS
LIN {X -16.287,Y -44.160,Z -110.495,A -90.000,B 90.000,C 0.000} C_DIS
LIN {X -16.345,Y -44.160,Z -110.348,A -90.000,B 90.000,C 0.000} C_DIS
LIN {X -17.120,Y -44.139,Z -108.890,A -90.000,B 90.000,C 0.000} C_DIS
LIN {X -17.167,Y -44.136,Z -108.799,A -90.000,B 90.000,C 0.000} C_DIS
LIN {X -17.289,Y -44.130,Z -108.549,A -90.000,B 90.000,C 0.000} C_DIS
LIN {X -17.438,Y -44.123,Z -108.213,A -90.000,B 90.000,C 0.000} C_DIS
LIN {X -17.512,Y -44.121,Z -108.037,A -90.000,B 90.000,C 0.000} C_DIS
LIN {X -17.678,Y -44.118,Z -107.601,A -90.000,B 90.000,C 0.000} C_DIS
LIN {X -18.405,Y -44.107,Z -105.524,A -90.000,B 90.000,C 0.000} C_DIS
LIN {X -18.513,Y -44.107,Z -105.208,A -90.000,B 90.000,C 0.000} C_DIS
LIN {X -18.580,Y -44.108,Z -104.998,A -90.000,B 90.000,C 0.000} C_DIS
LIN {X -18.749,Y -44.113,Z -104.392,A -90.000,B 90.000,C 0.000} C_DIS
LIN {X -18.972,Y -44.111,Z -103.577,A -90.000,B 90.000,C 0.000} C_DIS
LIN {X -19.030,Y -44.112,Z -103.332,A -90.000,B 90.000,C 0.000} C_DIS
LIN {X -19.101,Y -44.114,Z -102.981,A -90.000,B 90.000,C 0.000} C_DIS
LIN {X -19.142,Y -44.117,Z -102.735,A -90.000,B 90.000,C 0.000} C_DIS
LIN {X -19.156,Y -44.117,Z -102.623,A -90.000,B 90.000,C 0.000} C_DIS
LIN {X -19.255,Y -44.117,Z -101.784,A -90.000,B 90.000,C 0.000} C_DIS
LIN {X -19.317,Y -44.114,Z -101.252,A -90.000,B 90.000,C 0.000} C_DIS
LIN {X -19.373,Y -44.104,Z -100.752,A -90.000,B 90.000,C 0.000} C_DIS
LIN {X -19.398,Y -44.099,Z -100.630,A -90.000,B 90.000,C 0.000} C_DIS
LIN {X -19.420,Y -44.095,Z -100.511,A -90.000,B 90.000,C 0.000} C_DIS
LIN {X -19.476,Y -44.084,Z -100.163,A -90.000,B 90.000,C 0.000} C_DIS
LIN {X -19.494,Y -44.081,Z -100.036,A -90.000,B 90.000,C 0.000} C_DIS
LIN {X -19.527,Y -44.074,Z -99.729,A -90.000,B 90.000,C 0.000} C_DIS
LIN {X -19.554,Y -44.065,Z -99.330,A -90.000,B 90.000,C 0.000} C_DIS
LIN {X -19.563,Y -44.059,Z -99.066,A -90.000,B 90.000,C 0.000} C_DIS
LIN {X -19.564,Y -44.057,Z -98.940,A -90.000,B 90.000,C 0.000} C_DIS
LIN {X -19.561,Y -44.052,Z -98.624,A -90.000,B 90.000,C 0.000} C_DIS
LIN {X -19.556,Y -44.051,Z -98.481,A -90.000,B 90.000,C 0.000} C_DIS
LIN {X -19.541,Y -44.046,Z -98.274,A -90.000,B 90.000,C 0.000} C_DIS
LIN {X -19.518,Y -44.035,Z -98.008,A -90.000,B 90.000,C 0.000} C_DIS
LIN {X -19.490,Y -44.028,Z -97.808,A -90.000,B 90.000,C 0.000} C_DIS
LIN {X -19.424,Y -44.015,Z -97.383,A -90.000,B 90.000,C 0.000} C_DIS
LIN {X -19.388,Y -44.011,Z -97.205,A -90.000,B 90.000,C 0.000} C_DIS
LIN {X -19.284,Y -44.002,Z -96.756,A -90.000,B 90.000,C 0.000} C_DIS
LIN {X -19.234,Y -44.000,Z -96.564,A -90.000,B 90.000,C 0.000} C_DIS
LIN {X -19.042,Y -44.003,Z -95.907,A -90.000,B 90.000,C 0.000} C_DIS
LIN {X -18.991,Y -43.996,Z -95.736,A -90.000,B 90.000,C 0.000} C_DIS
LIN {X -18.667,Y -43.934,Z -94.671,A -90.000,B 90.000,C 0.000} C_DIS
LIN {X -18.546,Y -43.914,Z -94.307,A -90.000,B 90.000,C 0.000} C_DIS
LIN {X -18.469,Y -43.904,Z -94.099,A -90.000,B 90.000,C 0.000} C_DIS
LIN {X -18.338,Y -43.889,Z -93.746,A -90.000,B 90.000,C 0.000} C_DIS
LIN {X -18.287,Y -43.885,Z -93.616,A -90.000,B 90.000,C 0.000} C_DIS
LIN {X -18.191,Y -43.880,Z -93.386,A -90.000,B 90.000,C 0.000} C_DIS
LIN {X -18.169,Y -43.877,Z -93.337,A -90.000,B 90.000,C 0.000} C_DIS
LIN {X -18.052,Y -43.859,Z -93.089,A -90.000,B 90.000,C 0.000} C_DIS
LIN {X -17.947,Y -43.843,Z -92.887,A -90.000,B 90.000,C 0.000} C_DIS
LIN {X -17.811,Y -43.825,Z -92.640,A -90.000,B 90.000,C 0.000} C_DIS
LIN {X -17.663,Y -43.807,Z -92.386,A -90.000,B 90.000,C 0.000} C_DIS
LIN {X -17.541,Y -43.796,Z -92.194,A -90.000,B 90.000,C 0.000} C_DIS
LIN {X -17.345,Y -43.778,Z -91.896,A -90.000,B 90.000,C 0.000} C_DIS
LIN {X -17.256,Y -43.772,Z -91.769,A -90.000,B 90.000,C 0.000} C_DIS
LIN {X -17.095,Y -43.763,Z -91.557,A -90.000,B 90.000,C 0.000} C_DIS
LIN {X -16.952,Y -43.757,Z -91.382,A -90.000,B 90.000,C 0.000} C_DIS
LIN {X -16.860,Y -43.755,Z -91.270,A -90.000,B 90.000,C 0.000} C_DIS
LIN {X -16.689,Y -43.753,Z -91.073,A -90.000,B 90.000,C 0.000} C_DIS
LIN {X -16.497,Y -43.739,Z -90.859,A -90.000,B 90.000,C 0.000} C_DIS
LIN {X -16.364,Y -43.728,Z -90.714,A -90.000,B 90.000,C 0.000} C_DIS
LIN {X -15.286,Y -43.655,Z -89.592,A -90.000,B 90.000,C 0.000} C_DIS
LIN {X -15.217,Y -43.648,Z -89.508,A -90.000,B 90.000,C 0.000} C_DIS
LIN {X -15.035,Y -43.631,Z -89.302,A -90.000,B 90.000,C 0.000} C_DIS
LIN {X -14.820,Y -43.615,Z -89.076,A -90.000,B 90.000,C 0.000} C_DIS
LIN {X -14.601,Y -43.599,Z -88.857,A -90.000,B 90.000,C 0.000} C_DIS
LIN {X -14.323,Y -43.574,Z -88.600,A -90.000,B 90.000,C 0.000} C_DIS
LIN {X -14.186,Y -43.563,Z -88.482,A -90.000,B 90.000,C 0.000} C_DIS
LIN {X -13.980,Y -43.550,Z -88.314,A -90.000,B 90.000,C 0.000} C_DIS
LIN {X -13.747,Y -43.538,Z -88.138,A -90.000,B 90.000,C 0.000} C_DIS
LIN {X -13.453,Y -43.526,Z -87.931,A -90.000,B 90.000,C 0.000} C_DIS
LIN {X -13.278,Y -43.519,Z -87.816,A -90.000,B 90.000,C 0.000} C_DIS
LIN {X -12.710,Y -43.496,Z -87.474,A -90.000,B 90.000,C 0.000} C_DIS
LIN {X -12.375,Y -43.486,Z -87.286,A -90.000,B 90.000,C 0.000} C_DIS
LIN {X -11.670,Y -43.471,Z -86.923,A -90.000,B 90.000,C 0.000} C_DIS
LIN {X -11.053,Y -43.444,Z -86.611,A -90.000,B 90.000,C 0.000} C_DIS
LIN {X -9.982,Y -43.362,Z -86.071,A -90.000,B 90.000,C 0.000} C_DIS
LIN {X -9.291,Y -43.308,Z -85.723,A -90.000,B 90.000,C 0.000} C_DIS
LIN {X -9.291,Y -60.000,Z -85.723,A -90.000,B 90.000,C 0.000} C_DIS
LIN {X -18.321,Y -60.000,Z -121.010,A -90.000,B 90.000,C 0.000} C_DIS
LIN {X -18.321,Y -43.308,Z -121.010,A -90.000,B 90.000,C 0.000} C_DIS
LIN {X -18.132,Y -43.366,Z -120.429,A -90.000,B 90.000,C 0.000} C_DIS
LIN {X -18.059,Y -43.391,Z -120.073,A -90.000,B 90.000,C 0.000} C_DIS
LIN {X -17.990,Y -43.415,Z -119.776,A -90.000,B 90.000,C 0.000} C_DIS
LIN {X -17.933,Y -43.437,Z -119.548,A -90.000,B 90.000,C 0.000} C_DIS
LIN {X -17.877,Y -43.457,Z -119.346,A -90.000,B 90.000,C 0.000} C_DIS
LIN {X -17.780,Y -43.490,Z -119.015,A -90.000,B 90.000,C 0.000} C_DIS
LIN {X -17.621,Y -43.540,Z -118.535,A -90.000,B 90.000,C 0.000} C_DIS
LIN {X -17.366,Y -43.617,Z -117.848,A -90.000,B 90.000,C 0.000} C_DIS
LIN {X -17.291,Y -43.656,Z -117.332,A -90.000,B 90.000,C 0.000} C_DIS
LIN {X -17.253,Y -43.674,Z -117.111,A -90.000,B 90.000,C 0.000} C_DIS
LIN {X -17.173,Y -43.710,Z -116.703,A -90.000,B 90.000,C 0.000} C_DIS
LIN {X -17.124,Y -43.731,Z -116.476,A -90.000,B 90.000,C 0.000} C_DIS
LIN {X -17.019,Y -43.767,Z -116.062,A -90.000,B 90.000,C 0.000} C_DIS
LIN {X -16.992,Y -43.788,Z -115.716,A -90.000,B 90.000,C 0.000} C_DIS
LIN {X -16.976,Y -43.798,Z -115.564,A -90.000,B 90.000,C 0.000} C_DIS
LIN {X -16.977,Y -43.804,Z -115.440,A -90.000,B 90.000,C 0.000} C_DIS
LIN {X -16.975,Y -43.815,Z -115.216,A -90.000,B 90.000,C 0.000} C_DIS
LIN {X -16.948,Y -43.850,Z -114.588,A -90.000,B 90.000,C 0.000} C_DIS
LIN {X -16.967,Y -43.850,Z -114.513,A -90.000,B 90.000,C 0.000} C_DIS
LIN {X -17.055,Y -43.855,Z -114.126,A -90.000,B 90.000,C 0.000} C_DIS
LIN {X -17.090,Y -43.859,Z -113.962,A -90.000,B 90.000,C 0.000} C_DIS
LIN {X -17.238,Y -43.858,Z -113.557,A -90.000,B 90.000,C 0.000} C_DIS
LIN {X -17.378,Y -43.860,Z -113.132,A -90.000,B 90.000,C 0.000} C_DIS
LIN {X -17.491,Y -43.863,Z -112.756,A -90.000,B 90.000,C 0.000} C_DIS
LIN {X -17.571,Y -43.859,Z -112.588,A -90.000,B 90.000,C 0.000} C_DIS
LIN {X -17.703,Y -43.855,Z -112.286,A -90.000,B 90.000,C 0.000} C_DIS
LIN {X -18.142,Y -43.848,Z -111.177,A -90.000,B 90.000,C 0.000} C_DIS
LIN {X -18.911,Y -43.799,Z -109.718,A -90.000,B 90.000,C 0.000} C_DIS
LIN {X -19.057,Y -43.791,Z -109.421,A -90.000,B 90.000,C 0.000} C_DIS
LIN {X -19.170,Y -43.786,Z -109.170,A -90.000,B 90.000,C 0.000} C_DIS
LIN {X -19.237,Y -43.783,Z -109.019,A -90.000,B 90.000,C 0.000} C_DIS
LIN {X -19.328,Y -43.779,Z -108.801,A -90.000,B 90.000,C 0.000} C_DIS
LIN {X -19.506,Y -43.775,Z -108.336,A -90.000,B 90.000,C 0.000} C_DIS
LIN {X -20.033,Y -43.777,Z -106.843,A -90.000,B 90.000,C 0.000} C_DIS
LIN {X -20.202,Y -43.776,Z -106.358,A -90.000,B 90.000,C 0.000} C_DIS
LIN {X -20.373,Y -43.774,Z -105.866,A -90.000,B 90.000,C 0.000} C_DIS
LIN {X -20.480,Y -43.775,Z -105.527,A -90.000,B 90.000,C 0.000} C_DIS
LIN {X -20.603,Y -43.771,Z -105.081,A -90.000,B 90.000,C 0.000} C_DIS
LIN {X -20.871,Y -43.757,Z -104.095,A -90.000,B 90.000,C 0.000} C_DIS
LIN {X -20.944,Y -43.754,Z -103.791,A -90.000,B 90.000,C 0.000} C_DIS
LIN {X -21.029,Y -43.750,Z -103.366,A -90.000,B 90.000,C 0.000} C_DIS
LIN {X -21.081,Y -43.747,Z -103.053,A -90.000,B 90.000,C 0.000} C_DIS
LIN {X -21.094,Y -43.747,Z -102.960,A -90.000,B 90.000,C 0.000} C_DIS
LIN {X -21.178,Y -43.747,Z -102.262,A -90.000,B 90.000,C 0.000} C_DIS
LIN {X -21.317,Y -43.743,Z -101.070,A -90.000,B 90.000,C 0.000} C_DIS
LIN {X -21.354,Y -43.739,Z -100.878,A -90.000,B 90.000,C 0.000} C_DIS
LIN {X -21.409,Y -43.735,Z -100.543,A -90.000,B 90.000,C 0.000} C_DIS
LIN {X -21.443,Y -43.731,Z -100.319,A -90.000,B 90.000,C 0.000} C_DIS
LIN {X -21.484,Y -43.722,Z -99.947,A -90.000,B 90.000,C 0.000} C_DIS
LIN {X -21.517,Y -43.709,Z -99.470,A -90.000,B 90.000,C 0.000} C_DIS
LIN {X -21.531,Y -43.700,Z -99.078,A -90.000,B 90.000,C 0.000} C_DIS
LIN {X -21.531,Y -43.699,Z -98.959,A -90.000,B 90.000,C 0.000} C_DIS
LIN {X -21.527,Y -43.692,Z -98.549,A -90.000,B 90.000,C 0.000} C_DIS
LIN {X -21.522,Y -43.690,Z -98.411,A -90.000,B 90.000,C 0.000} C_DIS
LIN {X -21.505,Y -43.688,Z -98.142,A -90.000,B 90.000,C 0.000} C_DIS
LIN {X -21.480,Y -43.687,Z -97.847,A -90.000,B 90.000,C 0.000} C_DIS
LIN {X -21.471,Y -43.687,Z -97.761,A -90.000,B 90.000,C 0.000} C_DIS
LIN {X -21.437,Y -43.679,Z -97.517,A -90.000,B 90.000,C 0.000} C_DIS
LIN {X -21.370,Y -43.657,Z -97.093,A -90.000,B 90.000,C 0.000} C_DIS
LIN {X -21.355,Y -43.653,Z -97.008,A -90.000,B 90.000,C 0.000} C_DIS
LIN {X -21.319,Y -43.646,Z -96.830,A -90.000,B 90.000,C 0.000} C_DIS
LIN {X -21.199,Y -43.628,Z -96.317,A -90.000,B 90.000,C 0.000} C_DIS
LIN {X -21.134,Y -43.620,Z -96.071,A -90.000,B 90.000,C 0.000} C_DIS
LIN {X -20.994,Y -43.610,Z -95.596,A -90.000,B 90.000,C 0.000} C_DIS
LIN {X -20.872,Y -43.597,Z -95.186,A -90.000,B 90.000,C 0.000} C_DIS
LIN {X -20.803,Y -43.586,Z -94.958,A -90.000,B 90.000,C 0.000} C_DIS
LIN {X -20.545,Y -43.527,Z -94.117,A -90.000,B 90.000,C 0.000} C_DIS
LIN {X -20.409,Y -43.500,Z -93.711,A -90.000,B 90.000,C 0.000} C_DIS
LIN {X -20.375,Y -43.494,Z -93.617,A -90.000,B 90.000,C 0.000} C_DIS
LIN {X -20.189,Y -43.462,Z -93.119,A -90.000,B 90.000,C 0.000} C_DIS
LIN {X -20.108,Y -43.450,Z -92.912,A -90.000,B 90.000,C 0.000} C_DIS
LIN {X -19.969,Y -43.430,Z -92.586,A -90.000,B 90.000,C 0.000} C_DIS
LIN {X -19.823,Y -43.405,Z -92.280,A -90.000,B 90.000,C 0.000} C_DIS
LIN {X -19.689,Y -43.383,Z -92.019,A -90.000,B 90.000,C 0.000} C_DIS
LIN {X -19.525,Y -43.360,Z -91.720,A -90.000,B 90.000,C 0.000} C_DIS
LIN {X -19.355,Y -43.340,Z -91.427,A -90.000,B 90.000,C 0.000} C_DIS
LIN {X -19.197,Y -43.324,Z -91.176,A -90.000,B 90.000,C 0.000} C_DIS
LIN {X -19.016,Y -43.308,Z -90.900,A -90.000,B 90.000,C 0.000} C_DIS
LIN {X -19.016,Y -60.000,Z -90.900,A -90.000,B 90.000,C 0.000} C_DIS
LIN {X -19.338,Y -60.000,Z -117.468,A -90.000,B 90.000,C 0.000} C_DIS
LIN {X -19.338,Y -43.308,Z -117.468,A -90.000,B 90.000,C 0.000} C_DIS
LIN {X -19.288,Y -43.325,Z -117.332,A -90.000,B 90.000,C 0.000} C_DIS
LIN {X -19.244,Y -43.349,Z -117.027,A -90.000,B 90.000,C 0.000} C_DIS
LIN {X -19.206,Y -43.366,Z -116.805,A -90.000,B 90.000,C 0.000} C_DIS
LIN {X -19.107,Y -43.409,Z -116.295,A -90.000,B 90.000,C 0.000} C_DIS
LIN {X -19.058,Y -43.428,Z -116.064,A -90.000,B 90.000,C 0.000} C_DIS
LIN {X -18.972,Y -43.462,Z -115.715,A -90.000,B 90.000,C 0.000} C_DIS
LIN {X -18.950,Y -43.481,Z -115.445,A -90.000,B 90.000,C 0.000} C_DIS
LIN {X -18.949,Y -43.497,Z -115.174,A -90.000,B 90.000,C 0.000} C_DIS
LIN {X -18.933,Y -43.522,Z -114.766,A -90.000,B 90.000,C 0.000} C_DIS
LIN {X -18.992,Y -43.527,Z -114.504,A -90.000,B 90.000,C 0.000} C_DIS
LIN {X -19.090,Y -43.526,Z -114.237,A -90.000,B 90.000,C 0.000} C_DIS
LIN {X -19.252,Y -43.526,Z -113.746,A -90.000,B 90.000,C 0.000} C_DIS
LIN {X -19.336,Y -43.527,Z -113.469,A -90.000,B 90.000,C 0.000} C_DIS
LIN {X -19.352,Y -43.527,Z -113.436,A -90.000,B 90.000,C 0.000} C_DIS
LIN {X -19.508,Y -43.520,Z -113.079,A -90.000,B 90.000,C 0.000} C_DIS
LIN {X -19.933,Y -43.508,Z -112.007,A -90.000,B 90.000,C 0.000} C_DIS
LIN {X -20.650,Y -43.462,Z -110.647,A -90.000,B 90.000,C 0.000} C_DIS
LIN {X -20.823,Y -43.452,Z -110.296,A -90.000,B 90.000,C 0.000} C_DIS
LIN {X -21.036,Y -43.442,Z -109.824,A -90.000,B 90.000,C 0.000} C_DIS
LIN {X -21.144,Y -43.438,Z -109.568,A -90.000,B 90.000,C 0.000} C_DIS
LIN {X -21.345,Y -43.433,Z -109.044,A -90.000,B 90.000,C 0.000} C_DIS
LIN {X -21.385,Y -43.432,Z -108.932,A -90.000,B 90.000,C 0.000} C_DIS
LIN {X -21.686,Y -43.431,Z -108.077,A -90.000,B 90.000,C 0.000} C_DIS
LIN {X -21.890,Y -43.423,Z -107.495,A -90.000,B 90.000,C 0.000} C_DIS
LIN {X -22.229,Y -43.399,Z -106.508,A -90.000,B 90.000,C 0.000} C_DIS
LIN {X -22.352,Y -43.393,Z -106.118,A -90.000,B 90.000,C 0.000} C_DIS
LIN {X -22.401,Y -43.392,Z -105.944,A -90.000,B 90.000,C 0.000} C_DIS
LIN {X -22.763,Y -43.371,Z -104.613,A -90.000,B 90.000,C 0.000} C_DIS
LIN {X -22.851,Y -43.368,Z -104.255,A -90.000,B 90.000,C 0.000} C_DIS
LIN {X -22.953,Y -43.367,Z -103.757,A -90.000,B 90.000,C 0.000} C_DIS
LIN {X -23.018,Y -43.369,Z -103.377,A -90.000,B 90.000,C 0.000} C_DIS
LIN {X -23.040,Y -43.370,Z -103.232,A -90.000,B 90.000,C 0.000} C_DIS
LIN {X -23.085,Y -43.376,Z -102.861,A -90.000,B 90.000,C 0.000} C_DIS
LIN {X -23.128,Y -43.377,Z -102.509,A -90.000,B 90.000,C 0.000} C_DIS
LIN {X -23.231,Y -43.374,Z -101.624,A -90.000,B 90.000,C 0.000} C_DIS
LIN {X -23.260,Y -43.371,Z -101.374,A -90.000,B 90.000,C 0.000} C_DIS
LIN {X -23.281,Y -43.364,Z -101.256,A -90.000,B 90.000,C 0.000} C_DIS
LIN {X -23.337,Y -43.346,Z -100.908,A -90.000,B 90.000,C 0.000} C_DIS
LIN {X -23.380,Y -43.331,Z -100.615,A -90.000,B 90.000,C 0.000} C_DIS
LIN {X -23.429,Y -43.313,Z -100.171,A -90.000,B 90.000,C 0.000} C_DIS
LIN {X -23.441,Y -43.308,Z -100.020,A -90.000,B 90.000,C 0.000} C_DIS
LIN {X -23.441,Y -43.308,Z -100.018,A -90.000,B 90.000,C 0.000} C_DIS
LIN {X -23.428,Y -43.308,Z -99.768,A -90.000,B 90.000,C 0.000} C_DIS
LIN {X -23.408,Y -43.308,Z -99.532,A -90.000,B 90.000,C 0.000} C_DIS
LIN {X -23.158,Y -43.308,Z -98.170,A -90.000,B 90.000,C 0.000} C_DIS
LIN {X -22.939,Y -43.308,Z -97.079,A -90.000,B 90.000,C 0.000} C_DIS
LIN {X -22.870,Y -43.308,Z -96.852,A -90.000,B 90.000,C 0.000} C_DIS
LIN {X -22.523,Y -43.308,Z -95.978,A -90.000,B 90.000,C 0.000} C_DIS
LIN {X -21.944,Y -43.308,Z -94.653,A -90.000,B 90.000,C 0.000} C_DIS
LIN {X -21.829,Y -43.308,Z -94.446,A -90.000,B 90.000,C 0.000} C_DIS
LIN {X -21.348,Y -43.308,Z -93.716,A -90.000,B 90.000,C 0.000} C_DIS
LIN {X -20.443,Y -43.308,Z -92.415,A -90.000,B 90.000,C 0.000} C_DIS
LIN {X -20.288,Y -43.308,Z -92.236,A -90.000,B 90.000,C 0.000} C_DIS
LIN {X -19.368,Y -43.308,Z -91.267,A -90.000,B 90.000,C 0.000} C_DIS
LIN {X -18.447,Y -43.308,Z -90.308,A -90.000,B 90.000,C 0.000} C_DIS
LIN {X -16.107,Y -43.308,Z -88.452,A -90.000,B 90.000,C 0.000} C_DIS
LIN {X -15.918,Y -43.308,Z -88.310,A -90.000,B 90.000,C 0.000} C_DIS
LIN {X -15.875,Y -43.308,Z -88.280,A -90.000,B 90.000,C 0.000} C_DIS
LIN {X -15.795,Y -43.308,Z -88.233,A -90.000,B 90.000,C 0.000} C_DIS
LIN {X -13.757,Y -43.308,Z -87.150,A -90.000,B 90.000,C 0.000} C_DIS
LIN {X -13.542,Y -43.308,Z -87.050,A -90.000,B 90.000,C 0.000} C_DIS
LIN {X -12.428,Y -43.308,Z -86.573,A -90.000,B 90.000,C 0.000} C_DIS
LIN {X -11.296,Y -43.308,Z -86.180,A -90.000,B 90.000,C 0.000} C_DIS
LIN {X -9.655,Y -43.308,Z -85.804,A -90.000,B 90.000,C 0.000} C_DIS
LIN {X -8.582,Y -43.308,Z -85.567,A -90.000,B 90.000,C 0.000} C_DIS
LIN {X -7.532,Y -43.308,Z -85.447,A -90.000,B 90.000,C 0.000} C_DIS
LIN {X -7.066,Y -43.308,Z -85.401,A -90.000,B 90.000,C 0.000} C_DIS
LIN {X -6.605,Y -43.308,Z -85.355,A -90.000,B 90.000,C 0.000} C_DIS
LIN {X -5.521,Y -43.308,Z -85.286,A -90.000,B 90.000,C 0.000} C_DIS
LIN {X -4.691,Y -43.308,Z -85.307,A -90.000,B 90.000,C 0.000} C_DIS
LIN {X -2.573,Y -43.308,Z -85.334,A -90.000,B 90.000,C 0.000} C_DIS
LIN {X -2.292,Y -43.308,Z -85.353,A -90.000,B 90.000,C 0.000} C_DIS
LIN {X 0.363,Y -43.308,Z -85.580,A -90.000,B 90.000,C 0.000} C_DIS
LIN {X 0.711,Y -43.308,Z -85.605,A -90.000,B 90.000,C 0.000} C_DIS
LIN {X 1.468,Y -43.308,Z -85.699,A -90.000,B 90.000,C 0.000} C_DIS
LIN {X 3.780,Y -43.308,Z -86.044,A -90.000,B 90.000,C 0.000} C_DIS
LIN {X 4.179,Y -43.308,Z -86.110,A -90.000,B 90.000,C 0.000} C_DIS
LIN {X 4.538,Y -43.308,Z -86.178,A -90.000,B 90.000,C 0.000} C_DIS
LIN {X 7.122,Y -43.308,Z -86.604,A -90.000,B 90.000,C 0.000} C_DIS
LIN {X 8.263,Y -43.308,Z -86.823,A -90.000,B 90.000,C 0.000} C_DIS
LIN {X 9.915,Y -43.308,Z -87.098,A -90.000,B 90.000,C 0.000} C_DIS
LIN {X 11.604,Y -43.308,Z -87.399,A -90.000,B 90.000,C 0.000} C_DIS
LIN {X 12.573,Y -43.308,Z -87.549,A -90.000,B 90.000,C 0.000} C_DIS
LIN {X 14.764,Y -43.308,Z -87.875,A -90.000,B 90.000,C 0.000} C_DIS
LIN {X 15.143,Y -43.308,Z -87.924,A -90.000,B 90.000,C 0.000} C_DIS
LIN {X 16.722,Y -43.308,Z -88.092,A -90.000,B 90.000,C 0.000} C_DIS
LIN {X 17.735,Y -43.308,Z -88.232,A -90.000,B 90.000,C 0.000} C_DIS
LIN {X 17.953,Y -43.308,Z -88.259,A -90.000,B 90.000,C 0.000} C_DIS
LIN {X 20.166,Y -43.308,Z -88.467,A -90.000,B 90.000,C 0.000} C_DIS
LIN {X 21.059,Y -43.308,Z -88.503,A -90.000,B 90.000,C 0.000} C_DIS
LIN {X 22.819,Y -43.308,Z -88.618,A -90.000,B 90.000,C 0.000} C_DIS
LIN {X 24.685,Y -43.308,Z -88.588,A -90.000,B 90.000,C 0.000} C_DIS
LIN {X 25.115,Y -43.308,Z -88.613,A -90.000,B 90.000,C 0.000} C_DIS
LIN {X 25.493,Y -43.308,Z -88.600,A -90.000,B 90.000,C 0.000} C_DIS
LIN {X 28.146,Y -43.308,Z -88.540,A -90.000,B 90.000,C 0.000} C_DIS
LIN {X 28.302,Y -43.308,Z -88.519,A -90.000,B 90.000,C 0.000} C_DIS
LIN {X 28.582,Y -43.308,Z -88.488,A -90.000,B 90.000,C 0.000} C_DIS
LIN {X 31.525,Y -43.308,Z -88.518,A -90.000,B 90.000,C 0.000} C_DIS
LIN {X 32.521,Y -43.308,Z -88.428,A -90.000,B 90.000,C 0.000} C_DIS
LIN {X 32.758,Y -43.308,Z -88.426,A -90.000,B 90.000,C 0.000} C_DIS
LIN {X 34.060,Y -43.308,Z -88.497,A -90.000,B 90.000,C 0.000} C_DIS
LIN {X 36.144,Y -43.308,Z -88.927,A -90.000,B 90.000,C 0.000} C_DIS
LIN {X 36.444,Y -43.308,Z -88.967,A -90.000,B 90.000,C 0.000} C_DIS
LIN {X 36.668,Y -43.308,Z -89.013,A -90.000,B 90.000,C 0.000} C_DIS
LIN {X 36.790,Y -43.308,Z -89.044,A -90.000,B 90.000,C 0.000} C_DIS
LIN {X 38.743,Y -43.308,Z -89.659,A -90.000,B 90.000,C 0.000} C_DIS
LIN {X 38.958,Y -43.308,Z -89.753,A -90.000,B 90.000,C 0.000} C_DIS
LIN {X 40.501,Y -43.308,Z -90.484,A -90.000,B 90.000,C 0.000} C_DIS
LIN {X 40.877,Y -43.308,Z -90.695,A -90.000,B 90.000,C 0.000} C_DIS
LIN {X 41.069,Y -43.308,Z -90.832,A -90.000,B 90.000,C 0.000} C_DIS
LIN {X 41.325,Y -43.308,Z -91.025,A -90.000,B 90.000,C 0.000} C_DIS
LIN {X 42.714,Y -43.308,Z -91.802,A -90.000,B 90.000,C 0.000} C_DIS
LIN {X 42.771,Y -43.308,Z -91.843,A -90.000,B 90.000,C 0.000} C_DIS
LIN {X 42.905,Y -43.308,Z -91.939,A -90.000,B 90.000,C 0.000} C_DIS
LIN {X 43.826,Y -43.308,Z -92.616,A -90.000,B 90.000,C 0.000} C_DIS
LIN {X 44.623,Y -43.308,Z -93.280,A -90.000,B 90.000,C 0.000} C_DIS
LIN {X 45.573,Y -43.308,Z -94.329,A -90.000,B 90.000,C 0.000} C_DIS
LIN {X 46.134,Y -43.308,Z -94.869,A -90.000,B 90.000,C 0.000} C_DIS
LIN {X 46.293,Y -43.308,Z -95.044,A -90.000,B 90.000,C 0.000} C_DIS
LIN {X 46.673,Y -43.308,Z -95.522,A -90.000,B 90.000,C 0.000} C_DIS
LIN {X 46.793,Y -43.308,Z -95.727,A -90.000,B 90.000,C 0.000} C_DIS
LIN {X 48.550,Y -43.308,Z -98.805,A -90.000,B 90.000,C 0.000} C_DIS
LIN {X 48.871,Y -43.308,Z -99.550,A -90.000,B 90.000,C 0.000} C_DIS
LIN {X 49.085,Y -43.308,Z -100.188,A -90.000,B 90.000,C 0.000} C_DIS
LIN {X 49.159,Y -43.308,Z -100.460,A -90.000,B 90.000,C 0.000} C_DIS
LIN {X 49.771,Y -43.308,Z -103.000,A -90.000,B 90.000,C 0.000} C_DIS
LIN {X 50.106,Y -43.308,Z -106.776,A -90.000,B 90.000,C 0.000} C_DIS
LIN {X 50.102,Y -43.308,Z -107.241,A -90.000,B 90.000,C 0.000} C_DIS
LIN {X 50.096,Y -43.308,Z -107.369,A -90.000,B 90.000,C 0.000} C_DIS
LIN {X 50.041,Y -43.308,Z -107.771,A -90.000,B 90.000,C 0.000} C_DIS
LIN {X 49.653,Y -43.308,Z -111.174,A -90.000,B 90.000,C 0.000} C_DIS
LIN {X 49.606,Y -43.308,Z -111.452,A -90.000,B 90.000,C 0.000} C_DIS
LIN {X 48.908,Y -43.308,Z -114.351,A -90.000,B 90.000,C 0.000} C_DIS
LIN {X 48.720,Y -43.308,Z -115.189,A -90.000,B 90.000,C 0.000} C_DIS
LIN {X 48.611,Y -43.308,Z -115.488,A -90.000,B 90.000,C 0.000} C_DIS
LIN {X 47.994,Y -43.308,Z -117.170,A -90.000,B 90.000,C 0.000} C_DIS
LIN {X 47.351,Y -43.308,Z -118.906,A -90.000,B 90.000,C 0.000} C_DIS
LIN {X 47.242,Y -43.308,Z -119.152,A -90.000,B 90.000,C 0.000} C_DIS
LIN {X 46.979,Y -43.308,Z -119.641,A -90.000,B 90.000,C 0.000} C_DIS
LIN {X 45.325,Y -43.308,Z -122.524,A -90.000,B 90.000,C 0.000} C_DIS
LIN {X 45.152,Y -43.308,Z -122.792,A -90.000,B 90.000,C 0.000} C_DIS
LIN {X 43.361,Y -43.308,Z -125.034,A -90.000,B 90.000,C 0.000} C_DIS
LIN {X 42.661,Y -43.308,Z -125.870,A -90.000,B 90.000,C 0.000} C_DIS
LIN {X 42.573,Y -43.308,Z -125.973,A -90.000,B 90.000,C 0.000} C_DIS
LIN {X 39.928,Y -43.308,Z -128.606,A -90.000,B 90.000,C 0.000} C_DIS
LIN {X 39.674,Y -43.308,Z -128.849,A -90.000,B 90.000,C 0.000} C_DIS
LIN {X 39.571,Y -43.308,Z -128.944,A -90.000,B 90.000,C 0.000} C_DIS
LIN {X 37.870,Y -43.308,Z -130.413,A -90.000,B 90.000,C 0.000} C_DIS
LIN {X 36.649,Y -43.308,Z -131.460,A -90.000,B 90.000,C 0.000} C_DIS
LIN {X 36.582,Y -43.308,Z -131.520,A -90.000,B 90.000,C 0.000} C_DIS
LIN {X 33.610,Y -43.308,Z -133.902,A -90.000,B 90.000,C 0.000} C_DIS
LIN {X 31.341,Y -43.308,Z -135.714,A -90.000,B 90.000,C 0.000} C_DIS
LIN {X 30.810,Y -43.308,Z -136.190,A -90.000,B 90.000,C 0.000} C_DIS
LIN {X 29.143,Y -43.308,Z -137.443,A -90.000,B 90.000,C 0.000} C_DIS
LIN {X 27.981,Y -43.308,Z -138.410,A -90.000,B 90.000,C 0.000} C_DIS
LIN {X 27.674,Y -43.308,Z -138.632,A -90.000,B 90.000,C 0.000} C_DIS
LIN {X 25.928,Y -43.308,Z -139.785,A -90.000,B 90.000,C 0.000} C_DIS
LIN {X 24.687,Y -43.308,Z -140.663,A -90.000,B 90.000,C 0.000} C_DIS
LIN {X 24.496,Y -43.308,Z -140.770,A -90.000,B 90.000,C 0.000} C_DIS
LIN {X 23.229,Y -43.308,Z -141.440,A -90.000,B 90.000,C 0.000} C_DIS
LIN {X 21.307,Y -43.308,Z -142.487,A -90.000,B 90.000,C 0.000} C_DIS
LIN {X 20.942,Y -43.308,Z -142.657,A -90.000,B 90.000,C 0.000} C_DIS
LIN {X 18.481,Y -43.308,Z -143.584,A -90.000,B 90.000,C 0.000} C_DIS
LIN {X 17.125,Y -43.308,Z -144.089,A -90.000,B 90.000,C 0.000} C_DIS
LIN {X 16.867,Y -43.308,Z -144.181,A -90.000,B 90.000,C 0.000} C_DIS
LIN {X 16.646,Y -43.308,Z -144.238,A -90.000,B 90.000,C 0.000} C_DIS
LIN {X 13.896,Y -43.308,Z -144.940,A -90.000,B 90.000,C 0.000} C_DIS
LIN {X 12.487,Y -43.308,Z -145.288,A -90.000,B 90.000,C 0.000} C_DIS
LIN {X 12.011,Y -43.308,Z -145.379,A -90.000,B 90.000,C 0.000} C_DIS
LIN {X 9.292,Y -43.308,Z -145.793,A -90.000,B 90.000,C 0.000} C_DIS
LIN {X 7.531,Y -43.308,Z -146.039,A -90.000,B 90.000,C 0.000} C_DIS
LIN {X 7.154,Y -43.308,Z -146.078,A -90.000,B 90.000,C 0.000} C_DIS
LIN {X 3.167,Y -43.308,Z -146.205,A -90.000,B 90.000,C 0.000} C_DIS
LIN {X 2.837,Y -43.308,Z -146.209,A -90.000,B 90.000,C 0.000} C_DIS
LIN {X 2.488,Y -43.308,Z -146.200,A -90.000,B 90.000,C 0.000} C_DIS
LIN {X 2.401,Y -43.308,Z -146.192,A -90.000,B 90.000,C 0.000} C_DIS
LIN {X -1.543,Y -43.308,Z -145.709,A -90.000,B 90.000,C 0.000} C_DIS
LIN {X -1.916,Y -43.308,Z -145.647,A -90.000,B 90.000,C 0.000} C_DIS
LIN {X -5.495,Y -43.308,Z -144.614,A -90.000,B 90.000,C 0.000} C_DIS
LIN {X -5.864,Y -43.308,Z -144.510,A -90.000,B 90.000,C 0.000} C_DIS
LIN {X -6.191,Y -43.308,Z -144.382,A -90.000,B 90.000,C 0.000} C_DIS
LIN {X -8.276,Y -43.308,Z -143.408,A -90.000,B 90.000,C 0.000} C_DIS
LIN {X -9.641,Y -43.308,Z -142.727,A -90.000,B 90.000,C 0.000} C_DIS
LIN {X -9.810,Y -43.308,Z -142.631,A -90.000,B 90.000,C 0.000} C_DIS
LIN {X -9.931,Y -43.308,Z -142.555,A -90.000,B 90.000,C 0.000} C_DIS
LIN {X -10.929,Y -43.308,Z -141.835,A -90.000,B 90.000,C 0.000} C_DIS
LIN {X -12.903,Y -43.308,Z -140.317,A -90.000,B 90.000,C 0.000} C_DIS
LIN {X -13.142,Y -43.308,Z -140.106,A -90.000,B 90.000,C 0.000} C_DIS
LIN {X -14.289,Y -43.308,Z -138.891,A -90.000,B 90.000,C 0.000} C_DIS
LIN {X -14.493,Y -43.308,Z -138.645,A -90.000,B 90.000,C 0.000} C_DIS
LIN {X -15.645,Y -43.308,Z -137.164,A -90.000,B 90.000,C 0.000} C_DIS
LIN {X -15.759,Y -43.308,Z -136.997,A -90.000,B 90.000,C 0.000} C_DIS
LIN {X -15.913,Y -43.308,Z -136.737,A -90.000,B 90.000,C 0.000} C_DIS
LIN {X -15.922,Y -43.308,Z -136.722,A -90.000,B 90.000,C 0.000} C_DIS
LIN {X -15.971,Y -43.308,Z -136.633,A -90.000,B 90.000,C 0.000} C_DIS
LIN {X -16.480,Y -43.308,Z -135.679,A -90.000,B 90.000,C 0.000} C_DIS
LIN {X -16.936,Y -43.308,Z -134.588,A -90.000,B 90.000,C 0.000} C_DIS
LIN {X -17.023,Y -43.308,Z -134.320,A -90.000,B 90.000,C 0.000} C_DIS
LIN {X -17.232,Y -43.308,Z -133.437,A -90.000,B 90.000,C 0.000} C_DIS
LIN {X -17.485,Y -43.308,Z -132.481,A -90.000,B 90.000,C 0.000} C_DIS
LIN {X -17.656,Y -43.308,Z -131.236,A -90.000,B 90.000,C 0.000} C_DIS
LIN {X -17.696,Y -43.308,Z -130.782,A -90.000,B 90.000,C 0.000} C_DIS
LIN {X -17.720,Y -43.308,Z -130.250,A -90.000,B 90.000,C 0.000} C_DIS
LIN {X -17.683,Y -43.308,Z -129.660,A -90.000,B 90.000,C 0.000} C_DIS
LIN {X -17.742,Y -43.308,Z -128.261,A -90.000,B 90.000,C 0.000} C_DIS
LIN {X -17.761,Y -43.308,Z -127.083,A -90.000,B 90.000,C 0.000} C_DIS
LIN {X -17.699,Y -43.308,Z -126.231,A -90.000,B 90.000,C 0.000} C_DIS
LIN {X -17.640,Y -43.308,Z -125.109,A -90.000,B 90.000,C 0.000} C_DIS
LIN {X -17.725,Y -43.308,Z -124.342,A -90.000,B 90.000,C 0.000} C_DIS
LIN {X -17.871,Y -43.308,Z -123.619,A -90.000,B 90.000,C 0.000} C_DIS
LIN {X -18.460,Y -43.308,Z -120.204,A -90.000,B 90.000,C 0.000} C_DIS
LIN {X -18.699,Y -43.308,Z -119.424,A -90.000,B 90.000,C 0.000} C_DIS
LIN {X -19.587,Y -43.308,Z -116.705,A -90.000,B 90.000,C 0.000} C_DIS
LIN {X -19.949,Y -43.308,Z -115.528,A -90.000,B 90.000,C 0.000} C_DIS
LIN {X -20.152,Y -43.308,Z -114.920,A -90.000,B 90.000,C 0.000} C_DIS
LIN {X -21.125,Y -43.308,Z -111.933,A -90.000,B 90.000,C 0.000} C_DIS
LIN {X -22.106,Y -43.308,Z -108.978,A -90.000,B 90.000,C 0.000} C_DIS
LIN {X -22.257,Y -43.308,Z -108.443,A -90.000,B 90.000,C 0.000} C_DIS
LIN {X -22.660,Y -43.308,Z -106.621,A -90.000,B 90.000,C 0.000} C_DIS
LIN {X -22.875,Y -43.308,Z -105.716,A -90.000,B 90.000,C 0.000} C_DIS
LIN {X -23.100,Y -43.308,Z -104.559,A -90.000,B 90.000,C 0.000} C_DIS
LIN {X -23.468,Y -43.308,Z -102.674,A -90.000,B 90.000,C 0.000} C_DIS
LIN {X -23.489,Y -43.308,Z -102.536,A -90.000,B 90.000,C 0.000} C_DIS
LIN {X -23.505,Y -43.308,Z -102.406,A -90.000,B 90.000,C 0.000} C_DIS
LIN {X -23.543,Y -43.308,Z -101.992,A -90.000,B 90.000,C 0.000} C_DIS
LIN {X -23.441,Y -43.308,Z -100.018,A -90.000,B 90.000,C 0.000} C_DIS
LIN {X -23.441,Y -60.000,Z -100.018,A -90.000,B 90.000,C 0.000} C_DIS
LIN {X 38.808,Y -60.000,Z -210.497,A -90.000,B 90.000,C 0.000} C_DIS
LIN {X 38.808,Y -48.272,Z -210.497,A -90.000,B 90.000,C 0.000} C_DIS
LIN {X 38.681,Y -48.276,Z -210.745,A -90.000,B 90.000,C 0.000} C_DIS
LIN {X 38.468,Y -48.283,Z -211.146,A -90.000,B 90.000,C 0.000} C_DIS
LIN {X 37.367,Y -48.321,Z -213.704,A -90.000,B 90.000,C 0.000} C_DIS
LIN {X 37.211,Y -48.326,Z -214.037,A -90.000,B 90.000,C 0.000} C_DIS
LIN {X 36.978,Y -48.334,Z -214.484,A -90.000,B 90.000,C 0.000} C_DIS
LIN {X 36.466,Y -48.346,Z -215.407,A -90.000,B 90.000,C 0.000} C_DIS
LIN {X 36.159,Y -48.351,Z -215.960,A -90.000,B 90.000,C 0.000} C_DIS
LIN {X 35.353,Y -48.364,Z -217.647,A -90.000,B 90.000,C 0.000} C_DIS
LIN {X 35.169,Y -48.366,Z -217.998,A -90.000,B 90.000,C 0.000} C_DIS
LIN {X 34.285,Y -48.380,Z -219.578,A -90.000,B 90.000,C 0.000} C_DIS
LIN {X 33.592,Y -48.375,Z -220.822,A -90.000,B 90.000,C 0.000} C_DIS
LIN {X 32.931,Y -48.365,Z -222.127,A -90.000,B 90.000,C 0.000} C_DIS
LIN {X 31.500,Y -48.344,Z -224.749,A -90.000,B 90.000,C 0.000} C_DIS
LIN {X 30.982,Y -48.315,Z -225.703,A -90.000,B 90.000,C 0.000} C_DIS
LIN {X 30.293,Y -48.275,Z -227.046,A -90.000,B 90.000,C 0.000} C_DIS
LIN {X 30.923,Y -48.292,Z -226.517,A -90.000,B 90.000,C 0.000} C_DIS
LIN {X 32.152,Y -48.339,Z -224.900,A -90.000,B 90.000,C 0.000} C_DIS
LIN {X 33.581,Y -48.352,Z -223.014,A -90.000,B 90.000,C 0.000} C_DIS
LIN {X 34.086,Y -48.358,Z -222.053,A -90.000,B 90.000,C 0.000} C_DIS
LIN {X 35.223,Y -48.365,Z -219.886,A -90.000,B 90.000,C 0.000} C_DIS
LIN {X 35.654,Y -48.359,Z -219.064,A -90.000,B 90.000,C 0.000} C_DIS
LIN {X 35.674,Y -48.358,Z -219.027,A -90.000,B 90.000,C 0.000} C_DIS
LIN {X 35.712,Y -48.358,Z -218.958,A -90.000,B 90.000,C 0.000} C_DIS
LIN {X 36.860,Y -48.339,Z -216.021,A -90.000,B 90.000,C 0.000} C_DIS
LIN {X 37.133,Y -48.331,Z -215.321,A -90.000,B 90.000,C 0.000} C_DIS
LIN {X 37.496,Y -48.321,Z -214.448,A -90.000,B 90.000,C 0.000} C_DIS
LIN {X 38.480,Y -48.284,Z -211.442,A -90.000,B 90.000,C 0.000} C_DIS
LIN {X 38.808,Y -48.272,Z -210.497,A -90.000,B 90.000,C 0.000} C_DIS
LIN {X 38.689,Y -48.276,Z -210.746,A -90.000,B 90.000,C 0.000} C_DIS
LIN {X 38.576,Y -48.280,Z -210.995,A -90.000,B 90.000,C 0.000} C_DIS
LIN {X 38.511,Y -48.282,Z -211.153,A -90.000,B 90.000,C 0.000} C_DIS
LIN {X 38.481,Y -48.283,Z -211.252,A -90.000,B 90.000,C 0.000} C_DIS
LIN {X 38.409,Y -48.286,Z -211.519,A -90.000,B 90.000,C 0.000} C_DIS
LIN {X 38.347,Y -48.289,Z -211.789,A -90.000,B 90.000,C 0.000} C_DIS
LIN {X 38.294,Y -48.291,Z -212.063,A -90.000,B 90.000,C 0.000} C_DIS
LIN {X 38.271,Y -48.292,Z -212.201,A -90.000,B 90.000,C 0.000} C_DIS
LIN {X 38.232,Y -48.294,Z -212.479,A -90.000,B 90.000,C 0.000} C_DIS
LIN {X 38.187,Y -48.297,Z -212.902,A -90.000,B 90.000,C 0.000} C_DIS
LIN {X 38.167,Y -48.299,Z -213.187,A -90.000,B 90.000,C 0.000} C_DIS
LIN {X 38.153,Y -48.300,Z -213.475,A -90.000,B 90.000,C 0.000} C_DIS
LIN {X 38.145,Y -48.302,Z -213.764,A -90.000,B 90.000,C 0.000} C_DIS
LIN {X 38.135,Y -48.306,Z -214.710,A -90.000,B 90.000,C 0.000} C_DIS
LIN {X 38.104,Y -48.310,Z -215.793,A -90.000,B 90.000,C 0.000} C_DIS
LIN {X 38.084,Y -48.314,Z -216.958,A -90.000,B 90.000,C 0.000} C_DIS
LIN {X 38.066,Y -48.315,Z -217.392,A -90.000,B 90.000,C 0.000} C_DIS
LIN {X 38.045,Y -48.316,Z -217.679,A -90.000,B 90.000,C 0.000} C_DIS
LIN {X 38.017,Y -48.317,Z -217.962,A -90.000,B 90.000,C 0.000} C_DIS
LIN {X 37.980,Y -48.318,Z -218.243,A -90.000,B 90.000,C 0.000} C_DIS
LIN {X 37.932,Y -48.319,Z -218.520,A -90.000,B 90.000,C 0.000} C_DIS
LIN {X 37.904,Y -48.320,Z -218.657,A -90.000,B 90.000,C 0.000} C_DIS
LIN {X 37.839,Y -48.321,Z -218.927,A -90.000,B 90.000,C 0.000} C_DIS
LIN {X 37.801,Y -48.321,Z -219.061,A -90.000,B 90.000,C 0.000} C_DIS
LIN {X 37.716,Y -48.322,Z -219.324,A -90.000,B 90.000,C 0.000} C_DIS
LIN {X 37.666,Y -48.323,Z -219.452,A -90.000,B 90.000,C 0.000} C_DIS
LIN {X 37.527,Y -48.327,Z -219.809,A -90.000,B 90.000,C 0.000} C_DIS
LIN {X 37.425,Y -48.329,Z -219.994,A -90.000,B 90.000,C 0.000} C_DIS
LIN {X 37.139,Y -48.336,Z -220.539,A -90.000,B 90.000,C 0.000} C_DIS
LIN {X 35.267,Y -48.323,Z -224.105,A -90.000,B 90.000,C 0.000} C_DIS
LIN {X 35.164,Y -48.323,Z -224.236,A -90.000,B 90.000,C 0.000} C_DIS
LIN {X 34.379,Y -48.322,Z -225.273,A -90.000,B 90.000,C 0.000} C_DIS
LIN {X 34.073,Y -48.320,Z -225.677,A -90.000,B 90.000,C 0.000} C_DIS
LIN {X 32.380,Y -48.254,Z -227.905,A -90.000,B 90.000,C 0.000} C_DIS
LIN {X 30.380,Y -48.201,Z -229.584,A -90.000,B 90.000,C 0.000} C_DIS
LIN {X 29.698,Y -48.182,Z -230.153,A -90.000,B 90.000,C 0.000} C_DIS
LIN {X 28.168,Y -48.085,Z -231.459,A -90.000,B 90.000,C 0.000} C_DIS
LIN {X 27.683,Y -48.060,Z -231.767,A -90.000,B 90.000,C 0.000} C_DIS
LIN {X 27.436,Y -48.049,Z -231.916,A -90.000,B 90.000,C 0.000} C_DIS
LIN {X 25.949,Y -48.003,Z -232.426,A -90.000,B 90.000,C 0.000} C_DIS
LIN {X 26.434,Y -48.099,Z -230.845,A -90.000,B 90.000,C 0.000} C_DIS
LIN {X 26.578,Y -48.123,Z -230.375,A -90.000,B 90.000,C 0.000} C_DIS
LIN {X 26.841,Y -48.153,Z -229.519,A -90.000,B 90.000,C 0.000} C_DIS
LIN {X 26.943,Y -48.164,Z -229.275,A -90.000,B 90.000,C 0.000} C_DIS
LIN {X 27.047,Y -48.174,Z -229.060,A -90.000,B 90.000,C 0.000} C_DIS
LIN {X 27.530,Y -48.196,Z -228.054,A -90.000,B 90.000,C 0.000} C_DIS
LIN {X 27.777,Y -48.207,Z -227.571,A -90.000,B 90.000,C 0.000} C_DIS
LIN {X 28.026,Y -48.217,Z -227.086,A -90.000,B 90.000,C 0.000} C_DIS
LIN {X 29.203,Y -48.269,Z -224.789,A -90.000,B 90.000,C 0.000} C_DIS
LIN {X 29.687,Y -48.291,Z -223.897,A -90.000,B 90.000,C 0.000} C_DIS
LIN {X 30.178,Y -48.299,Z -222.997,A -90.000,B 90.000,C 0.000} C_DIS
LIN {X 31.176,Y -48.308,Z -221.169,A -90.000,B 90.000,C 0.000} C_DIS
LIN {X 31.828,Y -48.310,Z -219.881,A -90.000,B 90.000,C 0.000} C_DIS
LIN {X 32.379,Y -48.315,Z -218.893,A -90.000,B 90.000,C 0.000} C_DIS
LIN {X 32.863,Y -48.313,Z -218.026,A -90.000,B 90.000,C 0.000} C_DIS
LIN {X 33.423,Y -48.310,Z -217.023,A -90.000,B 90.000,C 0.000} C_DIS
LIN {X 33.580,Y -48.306,Z -216.723,A -90.000,B 90.000,C 0.000} C_DIS
LIN {X 34.381,Y -48.285,Z -215.044,A -90.000,B 90.000,C 0.000} C_DIS
LIN {X 35.230,Y -48.271,Z -213.515,A -90.000,B 90.000,C 0.000} C_DIS
LIN {X 35.407,Y -48.267,Z -213.175,A -90.000,B 90.000,C 0.000} C_DIS
LIN {X 35.530,Y -48.264,Z -212.913,A -90.000,B 90.000,C 0.000} C_DIS
LIN {X 35.995,Y -48.249,Z -211.835,A -90.000,B 90.000,C 0.000} C_DIS
LIN {X 36.664,Y -48.216,Z -210.281,A -90.000,B 90.000,C 0.000} C_DIS
LIN {X 36.916,Y -48.207,Z -209.806,A -90.000,B 90.000,C 0.000} C_DIS
LIN {X 37.052,Y -48.202,Z -209.541,A -90.000,B 90.000,C 0.000} C_DIS
LIN {X 37.089,Y -48.201,Z -209.464,A -90.000,B 90.000,C 0.000} C_DIS
LIN {X 37.174,Y -48.197,Z -209.278,A -90.000,B 90.000,C 0.000} C_DIS
LIN {X 37.245,Y -48.194,Z -209.115,A -90.000,B 90.000,C 0.000} C_DIS
LIN {X 37.360,Y -48.187,Z -208.827,A -90.000,B 90.000,C 0.000} C_DIS
LIN {X 37.993,Y -48.144,Z -207.056,A -90.000,B 90.000,C 0.000} C_DIS
LIN {X 38.274,Y -48.132,Z -206.266,A -90.000,B 90.000,C 0.000} C_DIS
LIN {X 38.549,Y -48.123,Z -205.607,A -90.000,B 90.000,C 0.000} C_DIS
LIN {X 38.660,Y -48.119,Z -205.327,A -90.000,B 90.000,C 0.000} C_DIS
LIN {X 38.756,Y -48.115,Z -205.060,A -90.000,B 90.000,C 0.000} C_DIS
LIN {X 38.977,Y -48.107,Z -204.497,A -90.000,B 90.000,C 0.000} C_DIS
LIN {X 39.493,Y -48.077,Z -203.185,A -90.000,B 90.000,C 0.000} C_DIS
LIN {X 39.889,Y -48.061,Z -202.179,A -90.000,B 90.000,C 0.000} C_DIS
LIN {X 40.020,Y -48.055,Z -201.818,A -90.000,B 90.000,C 0.000} C_DIS
LIN {X 40.104,Y -48.051,Z -201.561,A -90.000,B 90.000,C 0.000} C_DIS
LIN {X 40.169,Y -48.047,Z -201.327,A -90.000,B 90.000,C 0.000} C_DIS
LIN {X 40.257,Y -48.041,Z -200.970,A -90.000,B 90.000,C 0.000} C_DIS
LIN {X 40.314,Y -48.036,Z -200.702,A -90.000,B 90.000,C 0.000} C_DIS
LIN {X 40.360,Y -48.032,Z -200.446,A -90.000,B 90.000,C 0.000} C_DIS
LIN {X 40.507,Y -48.025,Z -200.059,A -90.000,B 90.000,C 0.000} C_DIS
LIN {X 40.657,Y -48.016,Z -199.664,A -90.000,B 90.000,C 0.000} C_DIS
LIN {X 40.902,Y -48.004,Z -199.019,A -90.000,B 90.000,C 0.000} C_DIS
LIN {X 40.940,Y -48.002,Z -198.912,A -90.000,B 90.000,C 0.000} C_DIS
LIN {X 40.957,Y -48.002,Z -198.865,A -90.000,B 90.000,C 0.000} C_DIS
LIN {X 41.055,Y -47.996,Z -198.561,A -90.000,B 90.000,C 0.000} C_DIS
LIN {X 41.102,Y -47.993,Z -198.397,A -90.000,B 90.000,C 0.000} C_DIS
LIN {X 41.228,Y -47.984,Z -197.900,A -90.000,B 90.000,C 0.000} C_DIS
LIN {X 41.273,Y -47.980,Z -197.705,A -90.000,B 90.000,C 0.000} C_DIS
LIN {X 41.322,Y -47.973,Z -197.449,A -90.000,B 90.000,C 0.000} C_DIS
LIN {X 41.351,Y -47.967,Z -197.278,A -90.000,B 90.000,C 0.000} C_DIS
LIN {X 41.430,Y -47.944,Z -196.690,A -90.000,B 90.000,C 0.000} C_DIS
LIN {X 41.540,Y -47.940,Z -196.437,A -90.000,B 90.000,C 0.000} C_DIS
LIN {X 41.656,Y -47.937,Z -196.144,A -90.000,B 90.000,C 0.000} C_DIS
LIN {X 41.797,Y -47.927,Z -195.737,A -90.000,B 90.000,C 0.000} C_DIS
LIN {X 41.869,Y -47.921,Z -195.514,A -90.000,B 90.000,C 0.000} C_DIS
LIN {X 41.920,Y -47.916,Z -195.338,A -90.000,B 90.000,C 0.000} C_DIS
LIN {X 42.221,Y -47.879,Z -194.134,A -90.000,B 90.000,C 0.000} C_DIS
LIN {X 42.761,Y -47.867,Z -193.253,A -90.000,B 90.000,C 0.000} C_DIS
LIN {X 42.955,Y -47.865,Z -192.939,A -90.000,B 90.000,C 0.000} C_DIS
LIN {X 43.193,Y -47.867,Z -192.689,A -90.000,B 90.000,C 0.000} C_DIS
LIN {X 43.599,Y -47.866,Z -192.264,A -90.000,B 90.000,C 0.000} C_DIS
LIN {X 43.767,Y -47.864,Z -192.079,A -90.000,B 90.000,C 0.000} C_DIS
LIN {X 43.964,Y -47.861,Z -191.852,A -90.000,B 90.000,C 0.000} C_DIS
LIN {X 44.049,Y -47.859,Z -191.747,A -90.000,B 90.000,C 0.000} C_DIS
LIN {X 44.725,Y -47.836,Z -190.897,A -90.000,B 90.000,C 0.000} C_DIS
LIN {X 44.822,Y -47.834,Z -190.808,A -90.000,B 90.000,C 0.000} C_DIS
LIN {X 45.015,Y -47.829,Z -190.623,A -90.000,B 90.000,C 0.000} C_DIS
LIN {X 45.311,Y -47.821,Z -190.316,A -90.000,B 90.000,C 0.000} C_DIS
LIN {X 45.520,Y -47.812,Z -190.085,A -90.000,B 90.000,C 0.000} C_DIS
LIN {X 45.534,Y -47.812,Z -190.069,A -90.000,B 90.000,C 0.000} C_DIS
LIN {X 45.968,Y -47.793,Z -189.544,A -90.000,B 90.000,C 0.000} C_DIS
LIN {X 45.973,Y -47.799,Z -189.758,A -90.000,B 90.000,C 0.000} C_DIS
LIN {X 45.947,Y -47.838,Z -191.164,A -90.000,B 90.000,C 0.000} C_DIS
LIN {X 45.848,Y -47.883,Z -192.915,A -90.000,B 90.000,C 0.000} C_DIS
LIN {X 45.808,Y -47.898,Z -193.631,A -90.000,B 90.000,C 0.000} C_DIS
LIN {X 45.783,Y -47.904,Z -193.919,A -90.000,B 90.000,C 0.000} C_DIS
LIN {X 45.766,Y -47.907,Z -194.025,A -90.000,B 90.000,C 0.000} C_DIS
LIN {X 45.585,Y -47.944,Z -195.331,A -90.000,B 90.000,C 0.000} C_DIS
LIN {X 45.259,Y -47.982,Z -196.688,A -90.000,B 90.000,C 0.000} C_DIS
LIN {X 44.907,Y -48.011,Z -197.909,A -90.000,B 90.000,C 0.000} C_DIS
LIN {X 44.064,Y -48.057,Z -200.831,A -90.000,B 90.000,C 0.000} C_DIS
LIN {X 43.921,Y -48.065,Z -201.294,A -90.000,B 90.000,C 0.000} C_DIS
LIN {X 43.068,Y -48.101,Z -203.982,A -90.000,B 90.000,C 0.000} C_DIS
LIN {X 42.643,Y -48.125,Z -205.320,A -90.000,B 90.000,C 0.000} C_DIS
LIN {X 41.980,Y -48.150,Z -207.362,A -90.000,B 90.000,C 0.000} C_DIS
LIN {X 41.812,Y -48.156,Z -207.867,A -90.000,B 90.000,C 0.000} C_DIS
LIN {X 41.055,Y -48.196,Z -210.121,A -90.000,B 90.000,C 0.000} C_DIS
LIN {X 40.369,Y -48.230,Z -212.098,A -90.000,B 90.000,C 0.000} C_DIS
LIN {X 39.756,Y -48.261,Z -213.970,A -90.000,B 90.000,C 0.000} C_DIS
LIN {X 39.372,Y -48.276,Z -215.144,A -90.000,B 90.000,C 0.000} C_DIS
LIN {X 38.980,Y -48.287,Z -216.089,A -90.000,B 90.000,C 0.000} C_DIS
LIN {X 37.666,Y -48.323,Z -219.452,A -90.000,B 90.000,C 0.000} C_DIS
LIN {X 37.534,Y -48.327,Z -219.814,A -90.000,B 90.000,C 0.000} C_DIS
LIN {X 37.461,Y -48.329,Z -219.964,A -90.000,B 90.000,C 0.000} C_DIS
LIN {X 37.367,Y -48.331,Z -220.179,A -90.000,B 90.000,C 0.000} C_DIS
LIN {X 37.307,Y -48.333,Z -220.324,A -90.000,B 90.000,C 0.000} C_DIS
LIN {X 37.194,Y -48.335,Z -220.617,A -90.000,B 90.000,C 0.000} C_DIS
LIN {X 37.141,Y -48.334,Z -220.765,A -90.000,B 90.000,C 0.000} C_DIS
LIN {X 37.040,Y -48.332,Z -221.062,A -90.000,B 90.000,C 0.000} C_DIS
LIN {X 36.947,Y -48.329,Z -221.363,A -90.000,B 90.000,C 0.000} C_DIS
LIN {X 36.860,Y -48.324,Z -221.666,A -90.000,B 90.000,C 0.000} C_DIS
LIN {X 36.741,Y -48.314,Z -222.124,A -90.000,B 90.000,C 0.000} C_DIS
LIN {X 36.667,Y -48.306,Z -222.432,A -90.000,B 90.000,C 0.000} C_DIS
LIN {X 36.597,Y -48.298,Z -222.742,A -90.000,B 90.000,C 0.000} C_DIS
LIN {X 36.468,Y -48.281,Z -223.365,A -90.000,B 90.000,C 0.000} C_DIS
LIN {X 36.258,Y -48.253,Z -224.462,A -90.000,B 90.000,C 0.000} C_DIS
LIN {X 36.151,Y -48.242,Z -224.878,A -90.000,B 90.000,C 0.000} C_DIS
LIN {X 36.138,Y -48.241,Z -224.913,A -90.000,B 90.000,C 0.000} C_DIS
LIN {X 35.821,Y -48.217,Z -225.769,A -90.000,B 90.000,C 0.000} C_DIS
LIN {X 35.653,Y -48.205,Z -226.193,A -90.000,B 90.000,C 0.000} C_DIS
LIN {X 35.535,Y -48.197,Z -226.474,A -90.000,B 90.000,C 0.000} C_DIS
LIN {X 35.412,Y -48.189,Z -226.752,A -90.000,B 90.000,C 0.000} C_DIS
LIN {X 35.215,Y -48.176,Z -227.165,A -90.000,B 90.000,C 0.000} C_DIS
LIN {X 35.076,Y -48.167,Z -227.437,A -90.000,B 90.000,C 0.000} C_DIS
LIN {X 35.003,Y -48.163,Z -227.572,A -90.000,B 90.000,C 0.000} C_DIS
LIN {X 34.852,Y -48.155,Z -227.839,A -90.000,B 90.000,C 0.000} C_DIS
LIN {X 34.773,Y -48.150,Z -227.971,A -90.000,B 90.000,C 0.000} C_DIS
LIN {X 34.608,Y -48.142,Z -228.233,A -90.000,B 90.000,C 0.000} C_DIS
LIN {X 34.522,Y -48.137,Z -228.362,A -90.000,B 90.000,C 0.000} C_DIS
LIN {X 34.342,Y -48.129,Z -228.618,A -90.000,B 90.000,C 0.000} C_DIS
LIN {X 34.248,Y -48.121,Z -228.744,A -90.000,B 90.000,C 0.000} C_DIS
LIN {X 33.836,Y -48.111,Z -229.286,A -90.000,B 90.000,C 0.000} C_DIS
LIN {X 33.116,Y -48.115,Z -229.894,A -90.000,B 90.000,C 0.000} C_DIS
LIN {X 31.640,Y -48.124,Z -231.135,A -90.000,B 90.000,C 0.000} C_DIS
LIN {X 31.446,Y -48.118,Z -231.298,A -90.000,B 90.000,C 0.000} C_DIS
LIN {X 30.968,Y -48.098,Z -231.696,A -90.000,B 90.000,C 0.000} C_DIS
LIN {X 30.152,Y -48.059,Z -232.393,A -90.000,B 90.000,C 0.000} C_DIS
LIN {X 29.360,Y -48.010,Z -233.069,A -90.000,B 90.000,C 0.000} C_DIS
LIN {X 28.736,Y -47.978,Z -233.465,A -90.000,B 90.000,C 0.000} C_DIS
LIN {X 28.291,Y -47.956,Z -233.735,A -90.000,B 90.000,C 0.000} C_DIS
LIN {X 27.839,Y -47.941,Z -233.890,A -90.000,B 90.000,C 0.000} C_DIS
LIN {X 25.697,Y -47.875,Z -234.624,A -90.000,B 90.000,C 0.000} C_DIS
LIN {X 24.400,Y -47.815,Z -235.066,A -90.000,B 90.000,C 0.000} C_DIS
LIN {X 23.868,Y -47.794,Z -235.248,A -90.000,B 90.000,C 0.000} C_DIS
LIN {X 23.411,Y -47.795,Z -235.163,A -90.000,B 90.000,C 0.000} C_DIS
LIN {X 23.295,Y -47.792,Z -235.141,A -90.000,B 90.000,C 0.000} C_DIS
LIN {X 23.575,Y -47.856,Z -233.683,A -90.000,B 90.000,C 0.000} C_DIS
LIN {X 23.750,Y -47.877,Z -232.782,A -90.000,B 90.000,C 0.000} C_DIS
LIN {X 23.933,Y -47.896,Z -232.187,A -90.000,B 90.000,C 0.000} C_DIS
LIN {X 24.965,Y -48.012,Z -228.836,A -90.000,B 90.000,C 0.000} C_DIS
LIN {X 25.125,Y -48.029,Z -228.452,A -90.000,B 90.000,C 0.000} C_DIS
LIN {X 25.198,Y -48.036,Z -228.300,A -90.000,B 90.000,C 0.000} C_DIS
LIN {X 25.754,Y -48.061,Z -227.145,A -90.000,B 90.000,C 0.000} C_DIS
LIN {X 26.251,Y -48.083,Z -226.173,A -90.000,B 90.000,C 0.000} C_DIS
LIN {X 26.749,Y -48.105,Z -225.203,A -90.000,B 90.000,C 0.000} C_DIS
LIN {X 27.450,Y -48.135,Z -223.836,A -90.000,B 90.000,C 0.000} C_DIS
LIN {X 27.806,Y -48.152,Z -223.179,A -90.000,B 90.000,C 0.000} C_DIS
LIN {X 29.425,Y -48.176,Z -220.212,A -90.000,B 90.000,C 0.000} C_DIS
LIN {X 30.065,Y -48.183,Z -218.944,A -90.000,B 90.000,C 0.000} C_DIS
LIN {X 30.476,Y -48.187,Z -218.206,A -90.000,B 90.000,C 0.000} C_DIS
LIN {X 31.681,Y -48.183,Z -216.050,A -90.000,B 90.000,C 0.000} C_DIS
LIN {X 31.806,Y -48.182,Z -215.807,A -90.000,B 90.000,C 0.000} C_DIS
LIN {X 32.605,Y -48.171,Z -214.131,A -90.000,B 90.000,C 0.000} C_DIS
LIN {X 32.936,Y -48.169,Z -213.532,A -90.000,B 90.000,C 0.000} C_DIS
LIN {X 33.483,Y -48.161,Z -212.547,A -90.000,B 90.000,C 0.000} C_DIS
LIN {X 33.605,Y -48.158,Z -212.314,A -90.000,B 90.000,C 0.000} C_DIS
LIN {X 33.696,Y -48.156,Z -212.122,A -90.000,B 90.000,C 0.000} C_DIS
LIN {X 33.913,Y -48.149,Z -211.620,A -90.000,B 90.000,C 0.000} C_DIS
LIN {X 34.861,Y -48.111,Z -209.417,A -90.000,B 90.000,C 0.000} C_DIS
LIN {X 35.164,Y -48.105,Z -208.847,A -90.000,B 90.000,C 0.000} C_DIS
LIN {X 35.272,Y -48.103,Z -208.635,A -90.000,B 90.000,C 0.000} C_DIS
LIN {X 35.357,Y -48.100,Z -208.449,A -90.000,B 90.000,C 0.000} C_DIS
LIN {X 35.409,Y -48.098,Z -208.329,A -90.000,B 90.000,C 0.000} C_DIS
LIN {X 35.478,Y -48.094,Z -208.154,A -90.000,B 90.000,C 0.000} C_DIS
LIN {X 35.888,Y -48.067,Z -207.009,A -90.000,B 90.000,C 0.000} C_DIS
LIN {X 36.410,Y -48.027,Z -205.547,A -90.000,B 90.000,C 0.000} C_DIS
LIN {X 36.717,Y -48.010,Z -204.814,A -90.000,B 90.000,C 0.000} C_DIS
LIN {X 36.799,Y -48.005,Z -204.603,A -90.000,B 90.000,C 0.000} C_DIS
LIN {X 36.824,Y -48.003,Z -204.534,A -90.000,B 90.000,C 0.000} C_DIS
LIN {X 36.883,Y -47.999,Z -204.366,A -90.000,B 90.000,C 0.000} C_DIS
LIN {X 37.118,Y -47.992,Z -203.769,A -90.000,B 90.000,C 0.000} C_DIS
LIN {X 38.039,Y -47.939,Z -201.428,A -90.000,B 90.000,C 0.000} C_DIS
LIN {X 38.126,Y -47.933,Z -201.187,A -90.000,B 90.000,C 0.000} C_DIS
LIN {X 38.169,Y -47.930,Z -201.060,A -90.000,B 90.000,C 0.000} C_DIS
LIN {X 38.199,Y -47.928,Z -200.963,A -90.000,B 90.000,C 0.000} C_DIS
LIN {X 38.245,Y -47.926,Z -200.796,A -90.000,B 90.000,C 0.000} C_DIS
LIN {X 38.317,Y -47.921,Z -200.500,A -90.000,B 90.000,C 0.000} C_DIS
LIN {X 38.360,Y -47.917,Z -200.294,A -90.000,B 90.000,C 0.000} C_DIS
LIN {X 38.424,Y -47.909,Z -199.920,A -90.000,B 90.000,C 0.000} C_DIS
LIN {X 38.522,Y -47.906,Z -199.663,A -90.000,B 90.000,C 0.000} C_DIS
LIN {X 39.042,Y -47.875,Z -198.297,A -90.000,B 90.000,C 0.000} C_DIS
LIN {X 39.079,Y -47.872,Z -198.188,A -90.000,B 90.000,C 0.000} C_DIS
LIN {X 39.151,Y -47.866,Z -197.963,A -90.000,B 90.000,C 0.000} C_DIS
LIN {X 39.184,Y -47.864,Z -197.844,A -90.000,B 90.000,C 0.000} C_DIS
LIN {X 39.293,Y -47.857,Z -197.412,A -90.000,B 90.000,C 0.000} C_DIS
LIN {X 39.314,Y -47.856,Z -197.318,A -90.000,B 90.000,C 0.000} C_DIS
LIN {X 39.361,Y -47.851,Z -197.074,A -90.000,B 90.000,C 0.000} C_DIS
LIN {X 39.380,Y -47.849,Z -196.960,A -90.000,B 90.000,C 0.000} C_DIS
LIN {X 39.487,Y -47.831,Z -196.152,A -90.000,B 90.000,C 0.000} C_DIS
LIN {X 39.709,Y -47.827,Z -195.642,A -90.000,B 90.000,C 0.000} C_DIS
LIN {X 39.787,Y -47.823,Z -195.440,A -90.000,B 90.000,C 0.000} C_DIS
LIN {X 39.922,Y -47.812,Z -195.049,A -90.000,B 90.000,C 0.000} C_DIS
LIN {X 39.965,Y -47.809,Z -194.912,A -90.000,B 90.000,C 0.000} C_DIS
LIN {X 39.997,Y -47.806,Z -194.800,A -90.000,B 90.000,C 0.000} C_DIS
LIN {X 40.356,Y -47.780,Z -193.354,A -90.000,B 90.000,C 0.000} C_DIS
LIN {X 40.913,Y -47.775,Z -192.445,A -90.000,B 90.000,C 0.000} C_DIS
LIN {X 41.232,Y -47.770,Z -191.925,A -90.000,B 90.000,C 0.000} C_DIS
LIN {X 41.279,Y -47.769,Z -191.851,A -90.000,B 90.000,C 0.000} C_DIS
LIN {X 41.377,Y -47.768,Z -191.700,A -90.000,B 90.000,C 0.000} C_DIS
LIN {X 42.153,Y -47.767,Z -190.886,A -90.000,B 90.000,C 0.000} C_DIS
LIN {X 42.288,Y -47.766,Z -190.736,A -90.000,B 90.000,C 0.000} C_DIS
LIN {X 42.462,Y -47.765,Z -190.534,A -90.000,B 90.000,C 0.000} C_DIS
LIN {X 43.259,Y -47.751,Z -189.530,A -90.000,B 90.000,C 0.000} C_DIS
LIN {X 43.474,Y -47.750,Z -189.334,A -90.000,B 90.000,C 0.000} C_DIS
LIN {X 43.624,Y -47.748,Z -189.188,A -90.000,B 90.000,C 0.000} C_DIS
LIN {X 43.870,Y -47.746,Z -188.932,A -90.000,B 90.000,C 0.000} C_DIS
LIN {X 44.029,Y -47.743,Z -188.754,A -90.000,B 90.000,C 0.000} C_DIS
LIN {X 45.160,Y -47.718,Z -187.382,A -90.000,B 90.000,C 0.000} C_DIS
LIN {X 46.237,Y -47.704,Z -186.367,A -90.000,B 90.000,C 0.000} C_DIS
LIN {X 46.441,Y -47.699,Z -186.176,A -90.000,B 90.000,C 0.000} C_DIS
LIN {X 46.598,Y -47.693,Z -186.026,A -90.000,B 90.000,C 0.000} C_DIS
LIN {X 46.790,Y -47.684,Z -185.830,A -90.000,B 90.000,C 0.000} C_DIS
LIN {X 46.923,Y -47.678,Z -185.685,A -90.000,B 90.000,C 0.000} C_DIS
LIN {X 47.463,Y -47.652,Z -185.037,A -90.000,B 90.000,C 0.000} C_DIS
LIN {X 47.892,Y -47.690,Z -186.704,A -90.000,B 90.000,C 0.000} C_DIS
LIN {X 47.902,Y -47.699,Z -187.055,A -90.000,B 90.000,C 0.000} C_DIS
LIN {X 47.951,Y -47.748,Z -188.756,A -90.000,B 90.000,C 0.000} C_DIS
LIN {X 47.973,Y -47.778,Z -189.755,A -90.000,B 90.000,C 0.000} C_DIS
LIN {X 47.954,Y -47.807,Z -190.773,A -90.000,B 90.000,C 0.000} C_DIS
LIN {X 47.946,Y -47.815,Z -191.204,A -90.000,B 90.000,C 0.000} C_DIS
LIN {X 47.946,Y -47.816,Z -191.238,A -90.000,B 90.000,C 0.000} C_DIS
LIN {X 47.802,Y -47.845,Z -193.767,A -90.000,B 90.000,C 0.000} C_DIS
LIN {X 47.767,Y -47.849,Z -194.178,A -90.000,B 90.000,C 0.000} C_DIS
LIN {X 47.738,Y -47.851,Z -194.353,A -90.000,B 90.000,C 0.000} C_DIS
LIN {X 47.551,Y -47.865,Z -195.705,A -90.000,B 90.000,C 0.000} C_DIS
LIN {X 47.190,Y -47.897,Z -197.200,A -90.000,B 90.000,C 0.000} C_DIS
LIN {X 47.136,Y -47.902,Z -197.391,A -90.000,B 90.000,C 0.000} C_DIS
LIN {X 46.673,Y -47.926,Z -198.994,A -90.000,B 90.000,C 0.000} C_DIS
LIN {X 45.979,Y -47.972,Z -201.401,A -90.000,B 90.000,C 0.000} C_DIS
LIN {X 45.800,Y -47.981,Z -201.983,A -90.000,B 90.000,C 0.000} C_DIS
LIN {X 45.621,Y -47.988,Z -202.545,A -90.000,B 90.000,C 0.000} C_DIS
LIN {X 44.545,Y -48.050,Z -205.933,A -90.000,B 90.000,C 0.000} C_DIS
LIN {X 44.404,Y -48.056,Z -206.367,A -90.000,B 90.000,C 0.000} C_DIS
LIN {X 43.880,Y -48.084,Z -207.981,A -90.000,B 90.000,C 0.000} C_DIS
LIN {X 43.812,Y -48.086,Z -208.190,A -90.000,B 90.000,C 0.000} C_DIS
LIN {X 42.946,Y -48.112,Z -210.768,A -90.000,B 90.000,C 0.000} C_DIS
LIN {X 42.255,Y -48.127,Z -212.754,A -90.000,B 90.000,C 0.000} C_DIS
LIN {X 41.244,Y -48.142,Z -215.840,A -90.000,B 90.000,C 0.000} C_DIS
LIN {X 40.822,Y -48.151,Z -216.856,A -90.000,B 90.000,C 0.000} C_DIS
LIN {X 40.764,Y -48.152,Z -217.003,A -90.000,B 90.000,C 0.000} C_DIS
LIN {X 39.334,Y -48.157,Z -220.659,A -90.000,B 90.000,C 0.000} C_DIS
LIN {X 39.168,Y -48.161,Z -220.960,A -90.000,B 90.000,C 0.000} C_DIS
LIN {X 38.987,Y -48.166,Z -221.305,A -90.000,B 90.000,C 0.000} C_DIS
LIN {X 38.132,Y -48.162,Z -222.935,A -90.000,B 90.000,C 0.000} C_DIS
LIN {X 36.947,Y -48.147,Z -225.192,A -90.000,B 90.000,C 0.000} C_DIS
LIN {X 36.731,Y -48.151,Z -225.468,A -90.000,B 90.000,C 0.000} C_DIS
LIN {X 35.969,Y -48.162,Z -226.476,A -90.000,B 90.000,C 0.000} C_DIS
LIN {X 35.010,Y -48.142,Z -227.741,A -90.000,B 90.000,C 0.000} C_DIS
LIN {X 34.248,Y -48.121,Z -228.744,A -90.000,B 90.000,C 0.000} C_DIS
LIN {X 34.189,Y -48.124,Z -228.824,A -90.000,B 90.000,C 0.000} C_DIS
LIN {X 34.079,Y -48.120,Z -228.988,A -90.000,B 90.000,C 0.000} C_DIS
LIN {X 33.977,Y -48.116,Z -229.158,A -90.000,B 90.000,C 0.000} C_DIS
LIN {X 33.889,Y -48.111,Z -229.323,A -90.000,B 90.000,C 0.000} C_DIS
LIN {X 33.765,Y -48.106,Z -229.486,A -90.000,B 90.000,C 0.000} C_DIS
LIN {X 33.601,Y -48.100,Z -229.725,A -90.000,B 90.000,C 0.000} C_DIS
LIN {X 33.451,Y -48.092,Z -229.973,A -90.000,B 90.000,C 0.000} C_DIS
LIN {X 33.312,Y -48.083,Z -230.230,A -90.000,B 90.000,C 0.000} C_DIS
LIN {X 33.225,Y -48.077,Z -230.406,A -90.000,B 90.000,C 0.000} C_DIS
LIN {X 33.141,Y -48.070,Z -230.584,A -90.000,B 90.000,C 0.000} C_DIS
LIN {X 32.981,Y -48.055,Z -230.947,A -90.000,B 90.000,C 0.000} C_DIS
LIN {X 32.754,Y -48.030,Z -231.499,A -90.000,B 90.000,C 0.000} C_DIS
LIN {X 32.603,Y -48.006,Z -231.868,A -90.000,B 90.000,C 0.000} C_DIS
LIN {X 32.447,Y -47.983,Z -232.232,A -90.000,B 90.000,C 0.000} C_DIS
LIN {X 32.324,Y -47.965,Z -232.501,A -90.000,B 90.000,C 0.000} C_DIS
LIN {X 32.237,Y -47.953,Z -232.677,A -90.000,B 90.000,C 0.000} C_DIS
LIN {X 32.148,Y -47.942,Z -232.850,A -90.000,B 90.000,C 0.000} C_DIS
LIN {X 32.054,Y -47.930,Z -233.020,A -90.000,B 90.000,C 0.000} C_DIS
LIN {X 31.955,Y -47.918,Z -233.188,A -90.000,B 90.000,C 0.000} C_DIS
LIN {X 31.852,Y -47.907,Z -233.351,A -90.000,B 90.000,C 0.000} C_DIS
LIN {X 31.742,Y -47.895,Z -233.510,A -90.000,B 90.000,C 0.000} C_DIS
LIN {X 31.626,Y -47.884,Z -233.664,A -90.000,B 90.000,C 0.000} C_DIS
LIN {X 31.502,Y -47.872,Z -233.811,A -90.000,B 90.000,C 0.000} C_DIS
LIN {X 31.370,Y -47.861,Z -233.953,A -90.000,B 90.000,C 0.000} C_DIS
LIN {X 31.229,Y -47.849,Z -234.089,A -90.000,B 90.000,C 0.000} C_DIS
LIN {X 31.155,Y -47.843,Z -234.154,A -90.000,B 90.000,C 0.000} C_DIS
LIN {X 30.580,Y -47.823,Z -234.647,A -90.000,B 90.000,C 0.000} C_DIS
LIN {X 30.516,Y -47.822,Z -234.694,A -90.000,B 90.000,C 0.000} C_DIS
LIN {X 29.815,Y -47.812,Z -235.141,A -90.000,B 90.000,C 0.000} C_DIS
LIN {X 29.147,Y -47.805,Z -235.548,A -90.000,B 90.000,C 0.000} C_DIS
LIN {X 28.294,Y -47.817,Z -235.845,A -90.000,B 90.000,C 0.000} C_DIS
LIN {X 28.017,Y -47.814,Z -235.941,A -90.000,B 90.000,C 0.000} C_DIS
LIN {X 27.705,Y -47.802,Z -236.047,A -90.000,B 90.000,C 0.000} C_DIS
LIN {X 24.346,Y -47.649,Z -237.193,A -90.000,B 90.000,C 0.000} C_DIS
LIN {X 23.979,Y -47.636,Z -237.297,A -90.000,B 90.000,C 0.000} C_DIS
LIN {X 22.102,Y -47.642,Z -236.948,A -90.000,B 90.000,C 0.000} C_DIS
LIN {X 22.006,Y -47.640,Z -236.930,A -90.000,B 90.000,C 0.000} C_DIS
LIN {X 21.627,Y -47.613,Z -236.858,A -90.000,B 90.000,C 0.000} C_DIS
LIN {X 21.103,Y -47.598,Z -235.973,A -90.000,B 90.000,C 0.000} C_DIS
LIN {X 21.694,Y -47.732,Z -232.900,A -90.000,B 90.000,C 0.000} C_DIS
LIN {X 21.812,Y -47.746,Z -232.292,A -90.000,B 90.000,C 0.000} C_DIS
LIN {X 22.768,Y -47.845,Z -229.190,A -90.000,B 90.000,C 0.000} C_DIS
LIN {X 23.088,Y -47.872,Z -228.152,A -90.000,B 90.000,C 0.000} C_DIS
LIN {X 23.302,Y -47.889,Z -227.641,A -90.000,B 90.000,C 0.000} C_DIS
LIN {X 23.449,Y -47.896,Z -227.333,A -90.000,B 90.000,C 0.000} C_DIS
LIN {X 23.981,Y -47.905,Z -226.231,A -90.000,B 90.000,C 0.000} C_DIS
LIN {X 24.978,Y -47.929,Z -224.291,A -90.000,B 90.000,C 0.000} C_DIS
LIN {X 25.347,Y -47.938,Z -223.571,A -90.000,B 90.000,C 0.000} C_DIS
LIN {X 25.702,Y -47.947,Z -222.880,A -90.000,B 90.000,C 0.000} C_DIS
LIN {X 25.902,Y -47.953,Z -222.513,A -90.000,B 90.000,C 0.000} C_DIS
LIN {X 26.398,Y -47.960,Z -221.604,A -90.000,B 90.000,C 0.000} C_DIS
LIN {X 27.679,Y -47.968,Z -219.258,A -90.000,B 90.000,C 0.000} C_DIS
LIN {X 28.308,Y -47.966,Z -218.011,A -90.000,B 90.000,C 0.000} C_DIS
LIN {X 29.479,Y -47.975,Z -215.914,A -90.000,B 90.000,C 0.000} C_DIS
LIN {X 29.832,Y -47.974,Z -215.281,A -90.000,B 90.000,C 0.000} C_DIS
LIN {X 29.918,Y -47.973,Z -215.128,A -90.000,B 90.000,C 0.000} C_DIS
LIN {X 30.010,Y -47.972,Z -214.953,A -90.000,B 90.000,C 0.000} C_DIS
LIN {X 30.836,Y -47.949,Z -213.221,A -90.000,B 90.000,C 0.000} C_DIS
LIN {X 31.211,Y -47.945,Z -212.546,A -90.000,B 90.000,C 0.000} C_DIS
LIN {X 31.744,Y -47.948,Z -211.583,A -90.000,B 90.000,C 0.000} C_DIS
LIN {X 31.838,Y -47.948,Z -211.400,A -90.000,B 90.000,C 0.000} C_DIS
LIN {X 31.895,Y -47.947,Z -211.279,A -90.000,B 90.000,C 0.000} C_DIS
LIN {X 32.274,Y -47.937,Z -210.396,A -90.000,B 90.000,C 0.000} C_DIS
LIN {X 33.065,Y -47.899,Z -208.558,A -90.000,B 90.000,C 0.000} C_DIS
LIN {X 33.395,Y -47.892,Z -207.938,A -90.000,B 90.000,C 0.000} C_DIS
LIN {X 33.473,Y -47.890,Z -207.788,A -90.000,B 90.000,C 0.000} C_DIS
LIN {X 33.549,Y -47.887,Z -207.621,A -90.000,B 90.000,C 0.000} C_DIS
LIN {X 33.596,Y -47.884,Z -207.510,A -90.000,B 90.000,C 0.000} C_DIS
LIN {X 33.629,Y -47.882,Z -207.423,A -90.000,B 90.000,C 0.000} C_DIS
LIN {X 34.104,Y -47.845,Z -206.094,A -90.000,B 90.000,C 0.000} C_DIS
LIN {X 34.551,Y -47.830,Z -204.832,A -90.000,B 90.000,C 0.000} C_DIS
LIN {X 34.878,Y -47.825,Z -204.048,A -90.000,B 90.000,C 0.000} C_DIS
LIN {X 34.926,Y -47.824,Z -203.924,A -90.000,B 90.000,C 0.000} C_DIS
LIN {X 34.981,Y -47.822,Z -203.775,A -90.000,B 90.000,C 0.000} C_DIS
LIN {X 35.002,Y -47.821,Z -203.706,A -90.000,B 90.000,C 0.000} C_DIS
LIN {X 35.126,Y -47.818,Z -203.390,A -90.000,B 90.000,C 0.000} C_DIS
LIN {X 35.335,Y -47.808,Z -202.860,A -90.000,B 90.000,C 0.000} C_DIS
LIN {X 36.181,Y -47.790,Z -200.701,A -90.000,B 90.000,C 0.000} C_DIS
LIN {X 36.256,Y -47.788,Z -200.495,A -90.000,B 90.000,C 0.000} C_DIS
LIN {X 36.298,Y -47.786,Z -200.359,A -90.000,B 90.000,C 0.000} C_DIS
LIN {X 36.377,Y -47.779,Z -200.032,A -90.000,B 90.000,C 0.000} C_DIS
LIN {X 36.405,Y -47.776,Z -199.898,A -90.000,B 90.000,C 0.000} C_DIS
LIN {X 36.489,Y -47.762,Z -199.398,A -90.000,B 90.000,C 0.000} C_DIS
LIN {X 37.176,Y -47.736,Z -197.590,A -90.000,B 90.000,C 0.000} C_DIS
LIN {X 37.245,Y -47.731,Z -197.371,A -90.000,B 90.000,C 0.000} C_DIS
LIN {X 37.358,Y -47.719,Z -196.926,A -90.000,B 90.000,C 0.000} C_DIS
LIN {X 37.402,Y -47.712,Z -196.700,A -90.000,B 90.000,C 0.000} C_DIS
LIN {X 37.481,Y -47.689,Z -196.108,A -90.000,B 90.000,C 0.000} C_DIS
LIN {X 37.546,Y -47.683,Z -195.614,A -90.000,B 90.000,C 0.000} C_DIS
LIN {X 37.562,Y -47.683,Z -195.579,A -90.000,B 90.000,C 0.000} C_DIS
LIN {X 37.656,Y -47.686,Z -195.362,A -90.000,B 90.000,C 0.000} C_DIS
LIN {X 37.868,Y -47.681,Z -194.874,A -90.000,B 90.000,C 0.000} C_DIS
LIN {X 37.924,Y -47.678,Z -194.728,A -90.000,B 90.000,C 0.000} C_DIS
LIN {X 38.032,Y -47.672,Z -194.410,A -90.000,B 90.000,C 0.000} C_DIS
LIN {X 38.060,Y -47.670,Z -194.319,A -90.000,B 90.000,C 0.000} C_DIS
LIN {X 38.231,Y -47.652,Z -193.637,A -90.000,B 90.000,C 0.000} C_DIS
LIN {X 38.493,Y -47.641,Z -192.576,A -90.000,B 90.000,C 0.000} C_DIS
LIN {X 38.882,Y -47.650,Z -191.941,A -90.000,B 90.000,C 0.000} C_DIS
LIN {X 39.540,Y -47.644,Z -190.865,A -90.000,B 90.000,C 0.000} C_DIS
LIN {X 39.799,Y -47.643,Z -190.462,A -90.000,B 90.000,C 0.000} C_DIS
LIN {X 40.707,Y -47.650,Z -189.508,A -90.000,B 90.000,C 0.000} C_DIS
LIN {X 40.806,Y -47.650,Z -189.399,A -90.000,B 90.000,C 0.000} C_DIS
LIN {X 40.925,Y -47.650,Z -189.260,A -90.000,B 90.000,C 0.000} C_DIS
LIN {X 41.140,Y -47.650,Z -188.988,A -90.000,B 90.000,C 0.000} C_DIS
LIN {X 41.793,Y -47.641,Z -188.165,A -90.000,B 90.000,C 0.000} C_DIS
LIN {X 42.125,Y -47.644,Z -187.860,A -90.000,B 90.000,C 0.000} C_DIS
LIN {X 42.225,Y -47.645,Z -187.763,A -90.000,B 90.000,C 0.000} C_DIS
LIN {X 42.422,Y -47.645,Z -187.556,A -90.000,B 90.000,C 0.000} C_DIS
LIN {X 42.516,Y -47.645,Z -187.449,A -90.000,B 90.000,C 0.000} C_DIS
LIN {X 42.749,Y -47.644,Z -187.166,A -90.000,B 90.000,C 0.000} C_DIS
LIN {X 43.156,Y -47.636,Z -186.672,A -90.000,B 90.000,C 0.000} C_DIS
LIN {X 43.698,Y -47.623,Z -186.015,A -90.000,B 90.000,C 0.000} C_DIS
LIN {X 45.153,Y -47.604,Z -184.645,A -90.000,B 90.000,C 0.000} C_DIS
LIN {X 45.237,Y -47.603,Z -184.561,A -90.000,B 90.000,C 0.000} C_DIS
LIN {X 45.353,Y -47.600,Z -184.442,A -90.000,B 90.000,C 0.000} C_DIS
LIN {X 45.434,Y -47.599,Z -184.351,A -90.000,B 90.000,C 0.000} C_DIS
LIN {X 46.080,Y -47.584,Z -183.573,A -90.000,B 90.000,C 0.000} C_DIS
LIN {X 46.847,Y -47.562,Z -182.630,A -90.000,B 90.000,C 0.000} C_DIS
LIN {X 46.942,Y -47.560,Z -182.506,A -90.000,B 90.000,C 0.000} C_DIS
LIN {X 47.369,Y -47.547,Z -181.921,A -90.000,B 90.000,C 0.000} C_DIS
LIN {X 47.905,Y -47.530,Z -181.183,A -90.000,B 90.000,C 0.000} C_DIS
LIN {X 48.309,Y -47.516,Z -180.593,A -90.000,B 90.000,C 0.000} C_DIS
LIN {X 48.787,Y -47.496,Z -179.864,A -90.000,B 90.000,C 0.000} C_DIS
LIN {X 48.791,Y -47.500,Z -180.002,A -90.000,B 90.000,C 0.000} C_DIS
LIN {X 48.815,Y -47.515,Z -180.748,A -90.000,B 90.000,C 0.000} C_DIS
LIN {X 48.824,Y -47.518,Z -180.886,A -90.000,B 90.000,C 0.000} C_DIS
LIN {X 48.843,Y -47.520,Z -181.059,A -90.000,B 90.000,C 0.000} C_DIS
LIN {X 48.857,Y -47.522,Z -181.154,A -90.000,B 90.000,C 0.000} C_DIS
LIN {X 48.888,Y -47.525,Z -181.343,A -90.000,B 90.000,C 0.000} C_DIS
LIN {X 48.967,Y -47.530,Z -181.736,A -90.000,B 90.000,C 0.000} C_DIS
LIN {X 49.057,Y -47.542,Z -182.481,A -90.000,B 90.000,C 0.000} C_DIS
LIN {X 49.187,Y -47.573,Z -183.574,A -90.000,B 90.000,C 0.000} C_DIS
LIN {X 49.204,Y -47.576,Z -183.688,A -90.000,B 90.000,C 0.000} C_DIS
LIN {X 49.257,Y -47.583,Z -183.970,A -90.000,B 90.000,C 0.000} C_DIS
LIN {X 49.285,Y -47.585,Z -184.096,A -90.000,B 90.000,C 0.000} C_DIS
LIN {X 49.532,Y -47.603,Z -185.059,A -90.000,B 90.000,C 0.000} C_DIS
LIN {X 49.821,Y -47.632,Z -186.177,A -90.000,B 90.000,C 0.000} C_DIS
LIN {X 49.884,Y -47.632,Z -186.426,A -90.000,B 90.000,C 0.000} C_DIS
LIN {X 49.919,Y -47.647,Z -187.664,A -90.000,B 90.000,C 0.000} C_DIS
LIN {X 49.949,Y -47.663,Z -188.715,A -90.000,B 90.000,C 0.000} C_DIS
LIN {X 49.971,Y -47.675,Z -189.754,A -90.000,B 90.000,C 0.000} C_DIS
LIN {X 49.941,Y -47.696,Z -191.315,A -90.000,B 90.000,C 0.000} C_DIS
LIN {X 49.846,Y -47.723,Z -193.003,A -90.000,B 90.000,C 0.000} C_DIS
LIN {X 49.795,Y -47.736,Z -193.895,A -90.000,B 90.000,C 0.000} C_DIS
LIN {X 49.750,Y -47.741,Z -194.427,A -90.000,B 90.000,C 0.000} C_DIS
LIN {X 49.708,Y -47.745,Z -194.681,A -90.000,B 90.000,C 0.000} C_DIS
LIN {X 49.562,Y -47.762,Z -195.745,A -90.000,B 90.000,C 0.000} C_DIS
LIN {X 49.516,Y -47.764,Z -196.078,A -90.000,B 90.000,C 0.000} C_DIS
LIN {X 49.121,Y -47.789,Z -197.713,A -90.000,B 90.000,C 0.000} C_DIS
LIN {X 48.921,Y -47.799,Z -198.407,A -90.000,B 90.000,C 0.000} C_DIS
LIN {X 48.146,Y -47.820,Z -201.088,A -90.000,B 90.000,C 0.000} C_DIS
LIN {X 47.885,Y -47.829,Z -201.993,A -90.000,B 90.000,C 0.000} C_DIS
LIN {X 47.700,Y -47.833,Z -202.590,A -90.000,B 90.000,C 0.000} C_DIS
LIN {X 47.069,Y -47.847,Z -204.570,A -90.000,B 90.000,C 0.000} C_DIS
LIN {X 46.441,Y -47.865,Z -206.545,A -90.000,B 90.000,C 0.000} C_DIS
LIN {X 45.697,Y -47.877,Z -208.825,A -90.000,B 90.000,C 0.000} C_DIS
LIN {X 44.824,Y -47.901,Z -211.422,A -90.000,B 90.000,C 0.000} C_DIS
LIN {X 44.134,Y -47.921,Z -213.409,A -90.000,B 90.000,C 0.000} C_DIS
LIN {X 43.696,Y -47.932,Z -214.748,A -90.000,B 90.000,C 0.000} C_DIS
LIN {X 43.111,Y -47.941,Z -216.532,A -90.000,B 90.000,C 0.000} C_DIS
LIN {X 42.659,Y -47.950,Z -217.621,A -90.000,B 90.000,C 0.000} C_DIS
LIN {X 41.140,Y -47.968,Z -221.508,A -90.000,B 90.000,C 0.000} C_DIS
LIN {X 40.910,Y -47.975,Z -221.925,A -90.000,B 90.000,C 0.000} C_DIS
LIN {X 38.626,Y -47.965,Z -226.279,A -90.000,B 90.000,C 0.000} C_DIS
LIN {X 38.297,Y -47.972,Z -226.699,A -90.000,B 90.000,C 0.000} C_DIS
LIN {X 37.933,Y -47.976,Z -227.180,A -90.000,B 90.000,C 0.000} C_DIS
LIN {X 35.289,Y -47.921,Z -230.665,A -90.000,B 90.000,C 0.000} C_DIS
LIN {X 33.774,Y -47.930,Z -231.943,A -90.000,B 90.000,C 0.000} C_DIS
LIN {X 32.246,Y -47.882,Z -233.219,A -90.000,B 90.000,C 0.000} C_DIS
LIN {X 31.155,Y -47.843,Z -234.154,A -90.000,B 90.000,C 0.000} C_DIS
LIN {X 31.051,Y -47.842,Z -234.245,A -90.000,B 90.000,C 0.000} C_DIS
LIN {X 30.849,Y -47.833,Z -234.433,A -90.000,B 90.000,C 0.000} C_DIS
LIN {X 30.606,Y -47.822,Z -234.679,A -90.000,B 90.000,C 0.000} C_DIS
LIN {X 30.555,Y -47.820,Z -234.726,A -90.000,B 90.000,C 0.000} C_DIS
LIN {X 30.244,Y -47.807,Z -234.994,A -90.000,B 90.000,C 0.000} C_DIS
LIN {X 30.044,Y -47.798,Z -235.180,A -90.000,B 90.000,C 0.000} C_DIS
LIN {X 29.750,Y -47.785,Z -235.466,A -90.000,B 90.000,C 0.000} C_DIS
LIN {X 29.559,Y -47.776,Z -235.661,A -90.000,B 90.000,C 0.000} C_DIS
LIN {X 29.394,Y -47.769,Z -235.836,A -90.000,B 90.000,C 0.000} C_DIS
LIN {X 29.164,Y -47.759,Z -236.019,A -90.000,B 90.000,C 0.000} C_DIS
LIN {X 28.965,Y -47.751,Z -236.187,A -90.000,B 90.000,C 0.000} C_DIS
LIN {X 28.562,Y -47.729,Z -236.510,A -90.000,B 90.000,C 0.000} C_DIS
LIN {X 27.374,Y -47.660,Z -237.502,A -90.000,B 90.000,C 0.000} C_DIS
LIN {X 26.971,Y -47.637,Z -237.826,A -90.000,B 90.000,C 0.000} C_DIS
LIN {X 26.766,Y -47.626,Z -237.984,A -90.000,B 90.000,C 0.000} C_DIS
LIN {X 26.453,Y -47.609,Z -238.214,A -90.000,B 90.000,C 0.000} C_DIS
LIN {X 26.132,Y -47.590,Z -238.433,A -90.000,B 90.000,C 0.000} C_DIS
LIN {X 25.912,Y -47.577,Z -238.573,A -90.000,B 90.000,C 0.000} C_DIS
LIN {X 25.800,Y -47.570,Z -238.640,A -90.000,B 90.000,C 0.000} C_DIS
LIN {X 25.573,Y -47.557,Z -238.770,A -90.000,B 90.000,C 0.000} C_DIS
LIN {X 25.339,Y -47.544,Z -238.892,A -90.000,B 90.000,C 0.000} C_DIS
LIN {X 25.100,Y -47.530,Z -239.005,A -90.000,B 90.000,C 0.000} C_DIS
LIN {X 24.947,Y -47.521,Z -239.073,A -90.000,B 90.000,C 0.000} C_DIS
LIN {X 24.724,Y -47.509,Z -239.152,A -90.000,B 90.000,C 0.000} C_DIS
LIN {X 24.462,Y -47.492,Z -239.233,A -90.000,B 90.000,C 0.000} C_DIS
LIN {X 24.082,Y -47.479,Z -239.344,A -90.000,B 90.000,C 0.000} C_DIS
LIN {X 21.189,Y -47.487,Z -238.806,A -90.000,B 90.000,C 0.000} C_DIS
LIN {X 20.992,Y -47.486,Z -238.785,A -90.000,B 90.000,C 0.000} C_DIS
LIN {X 20.816,Y -47.485,Z -238.775,A -90.000,B 90.000,C 0.000} C_DIS
LIN {X 20.658,Y -47.481,Z -238.766,A -90.000,B 90.000,C 0.000} C_DIS
LIN {X 20.432,Y -47.466,Z -238.752,A -90.000,B 90.000,C 0.000} C_DIS
LIN {X 20.253,Y -47.466,Z -238.449,A -90.000,B 90.000,C 0.000} C_DIS
LIN {X 19.000,Y -47.448,Z -236.337,A -90.000,B 90.000,C 0.000} C_DIS
LIN {X 19.509,Y -47.554,Z -233.696,A -90.000,B 90.000,C 0.000} C_DIS
LIN {X 19.695,Y -47.580,Z -232.726,A -90.000,B 90.000,C 0.000} C_DIS
LIN {X 19.794,Y -47.581,Z -232.225,A -90.000,B 90.000,C 0.000} C_DIS
LIN {X 19.863,Y -47.578,Z -231.874,A -90.000,B 90.000,C 0.000} C_DIS
LIN {X 19.884,Y -47.576,Z -231.779,A -90.000,B 90.000,C 0.000} C_DIS
LIN {X 20.014,Y -47.576,Z -231.361,A -90.000,B 90.000,C 0.000} C_DIS
LIN {X 21.226,Y -47.591,Z -227.469,A -90.000,B 90.000,C 0.000} C_DIS
LIN {X 21.498,Y -47.604,Z -226.824,A -90.000,B 90.000,C 0.000} C_DIS
LIN {X 21.531,Y -47.606,Z -226.755,A -90.000,B 90.000,C 0.000} C_DIS
LIN {X 22.210,Y -47.617,Z -225.347,A -90.000,B 90.000,C 0.000} C_DIS
LIN {X 23.219,Y -47.640,Z -223.383,A -90.000,B 90.000,C 0.000} C_DIS
LIN {X 23.953,Y -47.658,Z -221.953,A -90.000,B 90.000,C 0.000} C_DIS
LIN {X 24.057,Y -47.661,Z -221.762,A -90.000,B 90.000,C 0.000} C_DIS
LIN {X 25.942,Y -47.687,Z -218.308,A -90.000,B 90.000,C 0.000} C_DIS
LIN {X 26.559,Y -47.688,Z -217.082,A -90.000,B 90.000,C 0.000} C_DIS
LIN {X 28.189,Y -47.701,Z -214.161,A -90.000,B 90.000,C 0.000} C_DIS
LIN {X 28.249,Y -47.701,Z -214.044,A -90.000,B 90.000,C 0.000} C_DIS
LIN {X 29.071,Y -47.691,Z -212.315,A -90.000,B 90.000,C 0.000} C_DIS
LIN {X 30.009,Y -47.691,Z -210.622,A -90.000,B 90.000,C 0.000} C_DIS
LIN {X 30.072,Y -47.691,Z -210.499,A -90.000,B 90.000,C 0.000} C_DIS
LIN {X 31.197,Y -47.637,Z -207.884,A -90.000,B 90.000,C 0.000} C_DIS
LIN {X 31.275,Y -47.637,Z -207.703,A -90.000,B 90.000,C 0.000} C_DIS
LIN {X 31.445,Y -47.642,Z -207.381,A -90.000,B 90.000,C 0.000} C_DIS
LIN {X 31.679,Y -47.642,Z -206.940,A -90.000,B 90.000,C 0.000} C_DIS
LIN {X 31.740,Y -47.641,Z -206.804,A -90.000,B 90.000,C 0.000} C_DIS
LIN {X 31.773,Y -47.639,Z -206.718,A -90.000,B 90.000,C 0.000} C_DIS
LIN {X 32.622,Y -47.576,Z -204.338,A -90.000,B 90.000,C 0.000} C_DIS
LIN {X 32.699,Y -47.576,Z -204.121,A -90.000,B 90.000,C 0.000} C_DIS
LIN {X 33.045,Y -47.583,Z -203.286,A -90.000,B 90.000,C 0.000} C_DIS
LIN {X 33.092,Y -47.583,Z -203.161,A -90.000,B 90.000,C 0.000} C_DIS
LIN {X 33.126,Y -47.583,Z -203.052,A -90.000,B 90.000,C 0.000} C_DIS
LIN {X 33.184,Y -47.583,Z -202.904,A -90.000,B 90.000,C 0.000} C_DIS
LIN {X 34.016,Y -47.550,Z -200.787,A -90.000,B 90.000,C 0.000} C_DIS
LIN {X 34.334,Y -47.558,Z -199.971,A -90.000,B 90.000,C 0.000} C_DIS
LIN {X 34.380,Y -47.559,Z -199.838,A -90.000,B 90.000,C 0.000} C_DIS
LIN {X 34.443,Y -47.557,Z -199.573,A -90.000,B 90.000,C 0.000} C_DIS
LIN {X 34.559,Y -47.548,Z -198.879,A -90.000,B 90.000,C 0.000} C_DIS
LIN {X 34.619,Y -47.550,Z -198.720,A -90.000,B 90.000,C 0.000} C_DIS
LIN {X 35.014,Y -47.534,Z -197.682,A -90.000,B 90.000,C 0.000} C_DIS
LIN {X 35.314,Y -47.540,Z -196.886,A -90.000,B 90.000,C 0.000} C_DIS
LIN {X 35.426,Y -47.539,Z -196.441,A -90.000,B 90.000,C 0.000} C_DIS
LIN {X 35.606,Y -47.521,Z -195.077,A -90.000,B 90.000,C 0.000} C_DIS
LIN {X 35.686,Y -47.523,Z -194.892,A -90.000,B 90.000,C 0.000} C_DIS
LIN {X 36.035,Y -47.524,Z -194.090,A -90.000,B 90.000,C 0.000} C_DIS
LIN {X 36.142,Y -47.522,Z -193.772,A -90.000,B 90.000,C 0.000} C_DIS
LIN {X 36.294,Y -47.514,Z -193.160,A -90.000,B 90.000,C 0.000} C_DIS
LIN {X 36.631,Y -47.488,Z -191.800,A -90.000,B 90.000,C 0.000} C_DIS
LIN {X 36.861,Y -47.500,Z -191.421,A -90.000,B 90.000,C 0.000} C_DIS
LIN {X 36.948,Y -47.501,Z -191.279,A -90.000,B 90.000,C 0.000} C_DIS
LIN {X 37.843,Y -47.498,Z -189.818,A -90.000,B 90.000,C 0.000} C_DIS
LIN {X 38.223,Y -47.497,Z -189.225,A -90.000,B 90.000,C 0.000} C_DIS
LIN {X 38.840,Y -47.510,Z -188.575,A -90.000,B 90.000,C 0.000} C_DIS
LIN {X 39.263,Y -47.511,Z -188.132,A -90.000,B 90.000,C 0.000} C_DIS
LIN {X 39.361,Y -47.510,Z -188.021,A -90.000,B 90.000,C 0.000} C_DIS
LIN {X 40.329,Y -47.495,Z -186.801,A -90.000,B 90.000,C 0.000} C_DIS
LIN {X 40.779,Y -47.498,Z -186.389,A -90.000,B 90.000,C 0.000} C_DIS
LIN {X 40.976,Y -47.498,Z -186.182,A -90.000,B 90.000,C 0.000} C_DIS
LIN {X 42.070,Y -47.475,Z -184.855,A -90.000,B 90.000,C 0.000} C_DIS
LIN {X 42.228,Y -47.474,Z -184.662,A -90.000,B 90.000,C 0.000} C_DIS
LIN {X 42.256,Y -47.474,Z -184.634,A -90.000,B 90.000,C 0.000} C_DIS
LIN {X 43.373,Y -47.483,Z -183.579,A -90.000,B 90.000,C 0.000} C_DIS
LIN {X 43.783,Y -47.487,Z -183.193,A -90.000,B 90.000,C 0.000} C_DIS
LIN {X 43.867,Y -47.488,Z -183.108,A -90.000,B 90.000,C 0.000} C_DIS
LIN {X 43.921,Y -47.488,Z -183.048,A -90.000,B 90.000,C 0.000} C_DIS
LIN {X 44.499,Y -47.487,Z -182.352,A -90.000,B 90.000,C 0.000} C_DIS
LIN {X 44.857,Y -47.485,Z -181.910,A -90.000,B 90.000,C 0.000} C_DIS
LIN {X 45.294,Y -47.476,Z -181.372,A -90.000,B 90.000,C 0.000} C_DIS
LIN {X 45.357,Y -47.475,Z -181.290,A -90.000,B 90.000,C 0.000} C_DIS
LIN {X 46.255,Y -47.454,Z -180.055,A -90.000,B 90.000,C 0.000} C_DIS
LIN {X 46.660,Y -47.441,Z -179.465,A -90.000,B 90.000,C 0.000} C_DIS
LIN {X 47.463,Y -47.422,Z -178.236,A -90.000,B 90.000,C 0.000} C_DIS
LIN {X 47.834,Y -47.411,Z -177.667,A -90.000,B 90.000,C 0.000} C_DIS
LIN {X 47.960,Y -47.406,Z -177.468,A -90.000,B 90.000,C 0.000} C_DIS
LIN {X 48.160,Y -47.398,Z -177.135,A -90.000,B 90.000,C 0.000} C_DIS
LIN {X 48.486,Y -47.391,Z -176.587,A -90.000,B 90.000,C 0.000} C_DIS
LIN {X 48.626,Y -47.387,Z -176.360,A -90.000,B 90.000,C 0.000} C_DIS
LIN {X 49.270,Y -47.369,Z -175.316,A -90.000,B 90.000,C 0.000} C_DIS
LIN {X 49.508,Y -47.361,Z -174.906,A -90.000,B 90.000,C 0.000} C_DIS
LIN {X 49.984,Y -47.360,Z -174.608,A -90.000,B 90.000,C 0.000} C_DIS
LIN {X 49.981,Y -47.373,Z -175.133,A -90.000,B 90.000,C 0.000} C_DIS
LIN {X 50.023,Y -47.385,Z -175.551,A -90.000,B 90.000,C 0.000} C_DIS
LIN {X 50.099,Y -47.396,Z -175.917,A -90.000,B 90.000,C 0.000} C_DIS
LIN {X 50.192,Y -47.405,Z -176.364,A -90.000,B 90.000,C 0.000} C_DIS
LIN {X 50.448,Y -47.401,Z -177.598,A -90.000,B 90.000,C 0.000} C_DIS
LIN {X 50.529,Y -47.406,Z -177.987,A -90.000,B 90.000,C 0.000} C_DIS
LIN {X 50.576,Y -47.410,Z -178.326,A -90.000,B 90.000,C 0.000} C_DIS
LIN {X 50.637,Y -47.412,Z -178.575,A -90.000,B 90.000,C 0.000} C_DIS
LIN {X 50.692,Y -47.413,Z -178.727,A -90.000,B 90.000,C 0.000} C_DIS
LIN {X 50.709,Y -47.413,Z -178.768,A -90.000,B 90.000,C 0.000} C_DIS
LIN {X 50.777,Y -47.420,Z -179.537,A -90.000,B 90.000,C 0.000} C_DIS
LIN {X 50.798,Y -47.429,Z -180.257,A -90.000,B 90.000,C 0.000} C_DIS
LIN {X 50.812,Y -47.440,Z -180.684,A -90.000,B 90.000,C 0.000} C_DIS
LIN {X 50.819,Y -47.442,Z -180.761,A -90.000,B 90.000,C 0.000} C_DIS
LIN {X 50.848,Y -47.446,Z -180.951,A -90.000,B 90.000,C 0.000} C_DIS
LIN {X 50.942,Y -47.456,Z -181.420,A -90.000,B 90.000,C 0.000} C_DIS
LIN {X 51.090,Y -47.484,Z -182.646,A -90.000,B 90.000,C 0.000} C_DIS
LIN {X 51.172,Y -47.488,Z -183.340,A -90.000,B 90.000,C 0.000} C_DIS
LIN {X 51.220,Y -47.487,Z -183.601,A -90.000,B 90.000,C 0.000} C_DIS
LIN {X 51.683,Y -47.476,Z -185.411,A -90.000,B 90.000,C 0.000} C_DIS
LIN {X 51.872,Y -47.476,Z -186.148,A -90.000,B 90.000,C 0.000} C_DIS
LIN {X 51.913,Y -47.505,Z -187.610,A -90.000,B 90.000,C 0.000} C_DIS
LIN {X 51.942,Y -47.519,Z -188.626,A -90.000,B 90.000,C 0.000} C_DIS
LIN {X 51.966,Y -47.537,Z -189.753,A -90.000,B 90.000,C 0.000} C_DIS
LIN {X 51.939,Y -47.558,Z -191.182,A -90.000,B 90.000,C 0.000} C_DIS
LIN {X 51.935,Y -47.556,Z -191.394,A -90.000,B 90.000,C 0.000} C_DIS
LIN {X 51.782,Y -47.547,Z -194.025,A -90.000,B 90.000,C 0.000} C_DIS
LIN {X 51.727,Y -47.545,Z -194.676,A -90.000,B 90.000,C 0.000} C_DIS
LIN {X 51.671,Y -47.545,Z -195.010,A -90.000,B 90.000,C 0.000} C_DIS
LIN {X 51.471,Y -47.541,Z -196.450,A -90.000,B 90.000,C 0.000} C_DIS
LIN {X 51.042,Y -47.562,Z -198.224,A -90.000,B 90.000,C 0.000} C_DIS
